LIN {X 0,Y 354.943,Z 301.268,A -85,B 0,C 180,E1 -13486.255,E2 -13486.255} C_VEL
LIN {X 0,Y 354.946,Z 301.27,A -85,B 0,C 180,E1 -13489.735,E2 -13489.735} C_VEL
LIN {X 0,Y 355.073,Z 301.256,A -85,B 0,C 180,E1 -13493.18,E2 -13493.18} C_VEL
LIN {X 0,Y 355.22,Z 301.235,A -85,B 0,C 180,E1 -13497.732,E2 -13497.732} C_VEL
LIN {X 0,Y 355.215,Z 301.234,A -85,B 0,C 180,E1 -13502.268,E2 -13502.268} C_VEL
LIN {X 0,Y 355.075,Z 301.256,A -85,B 0,C 180,E1 -13506.82,E2 -13506.82} C_VEL
LIN {X 0,Y 354.946,Z 301.268,A -85,B 0,C 180,E1 -13510.265,E2 -13510.265} C_VEL
LIN {X 0,Y 354.934,Z 301.269,A -85,B 0,C 180,E1 -13514.019,E2 -13514.019} C_VEL
LIN {X 0,Y 354.881,Z 301.275,A -85,B 0,C 180,E1 -13518.093,E2 -13518.093} C_VEL
LIN {X 0,Y 354.807,Z 301.286,A -85,B 0,C 180,E1 -13522.108,E2 -13522.108} C_VEL
LIN {X 0,Y 354.856,Z 301.278,A -85,B 0,C 180,E1 -13525.831,E2 -13525.831} C_VEL
LIN {X 0,Y 354.8,Z 301.286,A -85,B 0,C 180,E1 -13529.684,E2 -13529.684} C_VEL
LIN {X 0,Y 354.808,Z 301.285,A -85,B 0,C 180,E1 -13533.685,E2 -13533.685} C_VEL
LIN {X 0,Y 354.791,Z 301.292,A -85,B 0,C 180,E1 -13536.46,E2 -13536.46} C_VEL
LIN {X 0,Y 354.818,Z 301.284,A -85,B 0,C 180,E1 -13539.425,E2 -13539.425} C_VEL
LIN {X 0,Y 354.782,Z 301.29,A -85,B 0,C 180,E1 -13542.868,E2 -13542.868} C_VEL
LIN {X 0,Y 354.762,Z 301.294,A -85,B 0,C 180,E1 -13546.105,E2 -13546.105} C_VEL
LIN {X 0,Y 354.783,Z 301.289,A -85,B 0,C 180,E1 -13549.18,E2 -13549.18} C_VEL
LIN {X 0,Y 354.803,Z 301.29,A -85,B 0,C 180,E1 -13552.404,E2 -13552.404} C_VEL
LIN {X 0,Y 354.808,Z 301.286,A -85,B 0,C 180,E1 -13554.942,E2 -13554.942} C_VEL
LIN {X 0,Y 354.791,Z 301.291,A -85,B 0,C 180,E1 -13558.406,E2 -13558.406} C_VEL
LIN {X 0,Y 354.845,Z 301.282,A -85,B 0,C 180,E1 -13561.62,E2 -13561.62} C_VEL
LIN {X 0,Y 354.898,Z 301.28,A -85,B 0,C 180,E1 -13564.174,E2 -13564.174} C_VEL
LIN {X 0,Y 354.845,Z 301.285,A -85,B 0,C 180,E1 -13567.283,E2 -13567.283} C_VEL
LIN {X 0,Y 356.535,Z 305.798,A -85,B 0,C 180,E1 -13567.509,E2 -13567.509} C_VEL
LIN {X 0,Y 362.776,Z 320.32,A -85,B 0,C 180,E1 -13568.226,E2 -13568.226} C_VEL
LIN {X 0,Y 363.979,Z 330.595,A -85,B 0,C 180,E1 -13568.518,E2 -13568.518} C_VEL
LIN {X 0,Y 362.433,Z 414.345,A -85,B 0,C 180,E1 -13570.201,E2 -13570.201} C_VEL
LIN {X 0,Y 361.996,Z 427.668,A -85,B 0,C 180,E1 -13570.693,E2 -13570.693} C_VEL
LIN {X 0,Y 361.185,Z 440.711,A -85,B 0,C 180,E1 -13571.421,E2 -13571.421} C_VEL
LIN {X 0,Y 360.332,Z 451.826,A -85,B 0,C 180,E1 -13572.258,E2 -13572.258} C_VEL
LIN {X 0,Y 359.319,Z 463.137,A -85,B 0,C 180,E1 -13573.356,E2 -13573.356} C_VEL
LIN {X 0,Y 358.318,Z 473.616,A -85,B 0,C 180,E1 -13574.647,E2 -13574.647} C_VEL
LIN {X 0,Y 357.214,Z 482.91,A -85,B 0,C 180,E1 -13576.055,E2 -13576.055} C_VEL
LIN {X 0,Y 356.336,Z 490.521,A -85,B 0,C 180,E1 -13577.471,E2 -13577.471} C_VEL
LIN {X 0,Y 355.47,Z 497.943,A -85,B 0,C 180,E1 -13579.175,E2 -13579.175} C_VEL
LIN {X 0,Y 354.666,Z 503.906,A -85,B 0,C 180,E1 -13580.88,E2 -13580.88} C_VEL
LIN {X 0,Y 354.158,Z 509.234,A -85,B 0,C 180,E1 -13582.848,E2 -13582.848} C_VEL
LIN {X 0,Y 353.853,Z 512.211,A -85,B 0,C 180,E1 -13584.302,E2 -13584.302} C_VEL
LIN {X 0,Y 353.61,Z 514.067,A -85,B 0,C 180,E1 -13585.441,E2 -13585.441} C_VEL
LIN {X 0,Y 353.524,Z 515.48,A -85,B 0,C 180,E1 -13586.582,E2 -13586.582} C_VEL
LIN {X 0,Y 353.413,Z 517.083,A -85,B 0,C 180,E1 -13588.862,E2 -13588.862} C_VEL
LIN {X 0,Y 353.399,Z 517.316,A -85,B 0,C 180,E1 -13590.001,E2 -13590.001} C_VEL
LIN {X 0,Y 353.413,Z 517.125,A -85,B 0,C 180,E1 -13591.141,E2 -13591.141} C_VEL
LIN {X 0,Y 353.52,Z 515.579,A -85,B 0,C 180,E1 -13593.42,E2 -13593.42} C_VEL
LIN {X 0,Y 353.604,Z 514.22,A -85,B 0,C 180,E1 -13594.561,E2 -13594.561} C_VEL
LIN {X 0,Y 353.952,Z 511.354,A -85,B 0,C 180,E1 -13596.271,E2 -13596.271} C_VEL
LIN {X 0,Y 354.266,Z 507.466,A -85,B 0,C 180,E1 -13597.983,E2 -13597.983} C_VEL
LIN {X 0,Y 354.854,Z 502.424,A -85,B 0,C 180,E1 -13599.693,E2 -13599.693} C_VEL
LIN {X 0,Y 355.657,Z 496.064,A -85,B 0,C 180,E1 -13601.398,E2 -13601.398} C_VEL
LIN {X 0,Y 356.581,Z 488.151,A -85,B 0,C 180,E1 -13603.101,E2 -13603.101} C_VEL
LIN {X 0,Y 357.641,Z 480.049,A -85,B 0,C 180,E1 -13604.511,E2 -13604.511} C_VEL
LIN {X 0,Y 358.795,Z 470.095,A -85,B 0,C 180,E1 -13605.917,E2 -13605.917} C_VEL
LIN {X 0,Y 359.629,Z 460.285,A -85,B 0,C 180,E1 -13607.047,E2 -13607.047} C_VEL
LIN {X 0,Y 360.561,Z 449.625,A -85,B 0,C 180,E1 -13608.026,E2 -13608.026} C_VEL
LIN {X 0,Y 361.45,Z 437.916,A -85,B 0,C 180,E1 -13608.861,E2 -13608.861} C_VEL
LIN {X 0,Y 362.145,Z 425.901,A -85,B 0,C 180,E1 -13609.485,E2 -13609.485} C_VEL
LIN {X 0,Y 362.603,Z 412.752,A -85,B 0,C 180,E1 -13609.939,E2 -13609.939} C_VEL
LIN {X 0,Y 363.133,Z 379.152,A -85,B 0,C 180,E1 -13610.626,E2 -13610.626} C_VEL
LIN {X 0,Y 362.558,Z 373.342,A -85,B 0,C 180,E1 -13610.782,E2 -13610.782} C_VEL
LIN {X 0,Y 357.516,Z 354.661,A -85,B 0,C 180,E1 -13611.489,E2 -13611.489} C_VEL
LIN {X 0,Y 357.093,Z 348.851,A -85,B 0,C 180,E1 -13611.64,E2 -13611.64} C_VEL
LIN {X 0,Y 357.337,Z 328.776,A -85,B 0,C 180,E1 -13612.052,E2 -13612.052} C_VEL
LIN {X 0,Y 356.257,Z 322.271,A -85,B 0,C 180,E1 -13612.263,E2 -13612.263} C_VEL
LIN {X 0,Y 347.959,Z 302.988,A -85,B 0,C 180,E1 -13613.254,E2 -13613.254} C_VEL
LIN {X 0,Y 347.823,Z 302.155,A -85,B 0,C 180,E1 -13613.286,E2 -13613.286} C_VEL
LIN {X 0,Y 347.855,Z 302.153,A -85,B 0,C 180,E1 -13617.255,E2 -13617.255} C_VEL
LIN {X 0,Y 347.765,Z 302.164,A -85,B 0,C 180,E1 -13620.347,E2 -13620.347} C_VEL
LIN {X 0,Y 347.749,Z 302.165,A -85,B 0,C 180,E1 -13624.465,E2 -13624.465} C_VEL
LIN {X 0,Y 347.781,Z 302.163,A -85,B 0,C 180,E1 -13627.99,E2 -13627.99} C_VEL
LIN {X 0,Y 347.756,Z 302.167,A -85,B 0,C 180,E1 -13631.831,E2 -13631.831} C_VEL
LIN {X 0,Y 347.772,Z 302.163,A -85,B 0,C 180,E1 -13635.017,E2 -13635.017} C_VEL
LIN {X 0,Y 347.755,Z 302.163,A -85,B 0,C 180,E1 -13638.398,E2 -13638.398} C_VEL
LIN {X 0,Y 347.779,Z 302.161,A -85,B 0,C 180,E1 -13642.012,E2 -13642.012} C_VEL
LIN {X 0,Y 347.75,Z 302.166,A -85,B 0,C 180,E1 -13645.536,E2 -13645.536} C_VEL
LIN {X 0,Y 347.75,Z 302.165,A -85,B 0,C 180,E1 -13648.301,E2 -13648.301} C_VEL
LIN {X 0,Y 347.784,Z 302.165,A -85,B 0,C 180,E1 -13650.988,E2 -13650.988} C_VEL
LIN {X 0,Y 347.836,Z 302.154,A -85,B 0,C 180,E1 -13653.608,E2 -13653.608} C_VEL
LIN {X 0,Y 347.84,Z 302.289,A -85,B 0,C 180,E1 -13657.347,E2 -13657.347} C_VEL
LIN {X 0,Y 348.699,Z 306.937,A -85,B 0,C 180,E1 -13658.715,E2 -13658.715} C_VEL
LIN {X 0,Y 352.108,Z 319.99,A -85,B 0,C 180,E1 -13659.233,E2 -13659.233} C_VEL
LIN {X 0,Y 354.168,Z 331.192,A -85,B 0,C 180,E1 -13659.635,E2 -13659.635} C_VEL
LIN {X 0,Y 351.818,Z 416.062,A -85,B 0,C 180,E1 -13662,E2 -13662} C_VEL
LIN {X 0,Y 351.384,Z 429.687,A -85,B 0,C 180,E1 -13662.616,E2 -13662.616} C_VEL
LIN {X 0,Y 350.662,Z 442.143,A -85,B 0,C 180,E1 -13663.405,E2 -13663.405} C_VEL
LIN {X 0,Y 350.051,Z 454.225,A -85,B 0,C 180,E1 -13664.407,E2 -13664.407} C_VEL
LIN {X 0,Y 349.42,Z 465.515,A -85,B 0,C 180,E1 -13665.587,E2 -13665.587} C_VEL
LIN {X 0,Y 348.563,Z 476.613,A -85,B 0,C 180,E1 -13667.038,E2 -13667.038} C_VEL
LIN {X 0,Y 347.87,Z 486.501,A -85,B 0,C 180,E1 -13668.64,E2 -13668.64} C_VEL
LIN {X 0,Y 347.315,Z 495.155,A -85,B 0,C 180,E1 -13670.39,E2 -13670.39} C_VEL
LIN {X 0,Y 346.876,Z 502.131,A -85,B 0,C 180,E1 -13672.139,E2 -13672.139} C_VEL
LIN {X 0,Y 346.533,Z 507.828,A -85,B 0,C 180,E1 -13673.954,E2 -13673.954} C_VEL
LIN {X 0,Y 346.411,Z 512.511,A -85,B 0,C 180,E1 -13675.928,E2 -13675.928} C_VEL
LIN {X 0,Y 346.281,Z 515.485,A -85,B 0,C 180,E1 -13677.674,E2 -13677.674} C_VEL
LIN {X 0,Y 346.265,Z 516.905,A -85,B 0,C 180,E1 -13678.837,E2 -13678.837} C_VEL
LIN {X 0,Y 346.291,Z 517.875,A -85,B 0,C 180,E1 -13680,E2 -13680} C_VEL
LIN {X 0,Y 346.374,Z 518.383,A -85,B 0,C 180,E1 -13681.163,E2 -13681.163} C_VEL
LIN {X 0,Y 346.512,Z 518.476,A -85,B 0,C 180,E1 -13682.325,E2 -13682.325} C_VEL
LIN {X 0,Y 346.709,Z 518.149,A -85,B 0,C 180,E1 -13683.486,E2 -13683.486} C_VEL
LIN {X 0,Y 346.782,Z 517.364,A -85,B 0,C 180,E1 -13684.65,E2 -13684.65} C_VEL
LIN {X 0,Y 346.874,Z 516.16,A -85,B 0,C 180,E1 -13685.814,E2 -13685.814} C_VEL
LIN {X 0,Y 347.646,Z 512.916,A -85,B 0,C 180,E1 -13687.864,E2 -13687.864} C_VEL
LIN {X 0,Y 348.502,Z 508.27,A -85,B 0,C 180,E1 -13689.87,E2 -13689.87} C_VEL
LIN {X 0,Y 349.62,Z 501.96,A -85,B 0,C 180,E1 -13691.891,E2 -13691.891} C_VEL
LIN {X 0,Y 350.753,Z 495.084,A -85,B 0,C 180,E1 -13693.617,E2 -13693.617} C_VEL
LIN {X 0,Y 352.112,Z 486.474,A -85,B 0,C 180,E1 -13695.335,E2 -13695.335} C_VEL
LIN {X 0,Y 353.615,Z 477.681,A -85,B 0,C 180,E1 -13696.749,E2 -13696.749} C_VEL
LIN {X 0,Y 355.127,Z 467.571,A -85,B 0,C 180,E1 -13698.083,E2 -13698.083} C_VEL
LIN {X 0,Y 356.807,Z 454.872,A -85,B 0,C 180,E1 -13699.413,E2 -13699.413} C_VEL
LIN {X 0,Y 358.181,Z 442.944,A -85,B 0,C 180,E1 -13700.382,E2 -13700.382} C_VEL
LIN {X 0,Y 359.347,Z 429.73,A -85,B 0,C 180,E1 -13701.212,E2 -13701.212} C_VEL
LIN {X 0,Y 360.302,Z 416.514,A -85,B 0,C 180,E1 -13701.791,E2 -13701.791} C_VEL
LIN {X 0,Y 365.349,Z 340.859,A -85,B 0,C 180,E1 -13704.251,E2 -13704.251} C_VEL
LIN {X 0,Y 363.993,Z 337.298,A -85,B 0,C 180,E1 -13704.591,E2 -13704.591} C_VEL
LIN {X 0,Y 358.725,Z 326.902,A -85,B 0,C 180,E1 -13705.835,E2 -13705.835} C_VEL
LIN {X 0,Y 353.588,Z 318.534,A -85,B 0,C 180,E1 -13707.102,E2 -13707.102} C_VEL
LIN {X 0,Y 351.324,Z 314.748,A -85,B 0,C 180,E1 -13707.724,E2 -13707.724} C_VEL
LIN {X 0,Y 350.188,Z 310.445,A -85,B 0,C 180,E1 -13710.346,E2 -13710.346} C_VEL
LIN {X 0,Y 349.155,Z 306.963,A -85,B 0,C 180,E1 -13712.92,E2 -13712.92} C_VEL
LIN {X 0,Y 348.281,Z 304.055,A -85,B 0,C 180,E1 -13715.817,E2 -13715.817} C_VEL
LIN {X 0,Y 347.734,Z 302.169,A -85,B 0,C 180,E1 -13718.795,E2 -13718.795} C_VEL
LIN {X 0,Y 347.743,Z 302.169,A -85,B 0,C 180,E1 -13721.831,E2 -13721.831} C_VEL
LIN {X 0,Y 347.742,Z 302.182,A -85,B 0,C 180,E1 -13725.42,E2 -13725.42} C_VEL
LIN {X 0,Y 348.287,Z 304.196,A -85,B 0,C 180,E1 -13728.298,E2 -13728.298} C_VEL
LIN {X 0,Y 348.856,Z 305.831,A -85,B 0,C 180,E1 -13729.955,E2 -13729.955} C_VEL
LIN {X 0,Y 350.413,Z 310.427,A -85,B 0,C 180,E1 -13733.346,E2 -13733.346} C_VEL
LIN {X 0,Y 351.765,Z 315.246,A -85,B 0,C 180,E1 -13735.983,E2 -13735.983} C_VEL
LIN {X 0,Y 353.418,Z 321.647,A -85,B 0,C 180,E1 -13738.866,E2 -13738.866} C_VEL
LIN {X 0,Y 354.923,Z 328.994,A -85,B 0,C 180,E1 -13741.624,E2 -13741.624} C_VEL
LIN {X 0,Y 355.421,Z 333.185,A -85,B 0,C 180,E1 -13743.008,E2 -13743.008} C_VEL
LIN {X 0,Y 358.864,Z 346.581,A -85,B 0,C 180,E1 -13744.17,E2 -13744.17} C_VEL
LIN {X 0,Y 361.513,Z 360.04,A -85,B 0,C 180,E1 -13745.139,E2 -13745.139} C_VEL
LIN {X 0,Y 363.058,Z 371.025,A -85,B 0,C 180,E1 -13745.804,E2 -13745.804} C_VEL
LIN {X 0,Y 363.51,Z 377.914,A -85,B 0,C 180,E1 -13746.146,E2 -13746.146} C_VEL
LIN {X 0,Y 359.161,Z 446.637,A -85,B 0,C 180,E1 -13748.362,E2 -13748.362} C_VEL
LIN {X 0,Y 357.866,Z 460.11,A -85,B 0,C 180,E1 -13748.997,E2 -13748.997} C_VEL
LIN {X 0,Y 356.387,Z 472.712,A -85,B 0,C 180,E1 -13749.811,E2 -13749.811} C_VEL
LIN {X 0,Y 354.63,Z 485.801,A -85,B 0,C 180,E1 -13750.913,E2 -13750.913} C_VEL
LIN {X 0,Y 352.739,Z 498.651,A -85,B 0,C 180,E1 -13752.31,E2 -13752.31} C_VEL
LIN {X 0,Y 351.199,Z 508.989,A -85,B 0,C 180,E1 -13753.729,E2 -13753.729} C_VEL
LIN {X 0,Y 349.796,Z 517.581,A -85,B 0,C 180,E1 -13755.156,E2 -13755.156} C_VEL
LIN {X 0,Y 348.612,Z 526.071,A -85,B 0,C 180,E1 -13756.89,E2 -13756.89} C_VEL
LIN {X 0,Y 347.626,Z 532.987,A -85,B 0,C 180,E1 -13758.63,E2 -13758.63} C_VEL
LIN {X 0,Y 346.843,Z 539.297,A -85,B 0,C 180,E1 -13760.67,E2 -13760.67} C_VEL
LIN {X 0,Y 346.405,Z 543.453,A -85,B 0,C 180,E1 -13762.421,E2 -13762.421} C_VEL
LIN {X 0,Y 346.23,Z 546.523,A -85,B 0,C 180,E1 -13764.174,E2 -13764.174} C_VEL
LIN {X 0,Y 346.181,Z 548.006,A -85,B 0,C 180,E1 -13765.341,E2 -13765.341} C_VEL
LIN {X 0,Y 346.167,Z 549.058,A -85,B 0,C 180,E1 -13766.507,E2 -13766.507} C_VEL
LIN {X 0,Y 346.159,Z 549.629,A -85,B 0,C 180,E1 -13767.672,E2 -13767.672} C_VEL
LIN {X 0,Y 346.29,Z 549.774,A -85,B 0,C 180,E1 -13768.836,E2 -13768.836} C_VEL
LIN {X 0,Y 346.36,Z 549.487,A -85,B 0,C 180,E1 -13769.999,E2 -13769.999} C_VEL
LIN {X 0,Y 346.289,Z 547.742,A -85,B 0,C 180,E1 -13772.325,E2 -13772.325} C_VEL
LIN {X 0,Y 346.22,Z 546.705,A -85,B 0,C 180,E1 -13773.49,E2 -13773.49} C_VEL
LIN {X 0,Y 346.251,Z 545.261,A -85,B 0,C 180,E1 -13774.656,E2 -13774.656} C_VEL
LIN {X 0,Y 346.281,Z 542.259,A -85,B 0,C 180,E1 -13776.407,E2 -13776.407} C_VEL
LIN {X 0,Y 346.488,Z 538.188,A -85,B 0,C 180,E1 -13778.161,E2 -13778.161} C_VEL
LIN {X 0,Y 346.933,Z 531.911,A -85,B 0,C 180,E1 -13780.209,E2 -13780.209} C_VEL
LIN {X 0,Y 347.597,Z 525.071,A -85,B 0,C 180,E1 -13781.96,E2 -13781.96} C_VEL
LIN {X 0,Y 348.436,Z 518.09,A -85,B 0,C 180,E1 -13783.411,E2 -13783.411} C_VEL
LIN {X 0,Y 349.454,Z 509.07,A -85,B 0,C 180,E1 -13784.947,E2 -13784.947} C_VEL
LIN {X 0,Y 350.467,Z 499.204,A -85,B 0,C 180,E1 -13786.303,E2 -13786.303} C_VEL
LIN {X 0,Y 351.59,Z 488.855,A -85,B 0,C 180,E1 -13787.447,E2 -13787.447} C_VEL
LIN {X 0,Y 352.712,Z 477.474,A -85,B 0,C 180,E1 -13788.439,E2 -13788.439} C_VEL
LIN {X 0,Y 353.77,Z 464.4,A -85,B 0,C 180,E1 -13789.284,E2 -13789.284} C_VEL
LIN {X 0,Y 354.594,Z 452.101,A -85,B 0,C 180,E1 -13789.84,E2 -13789.84} C_VEL
LIN {X 0,Y 355.014,Z 439.719,A -85,B 0,C 180,E1 -13790.193,E2 -13790.193} C_VEL
LIN {X 0,Y 356.114,Z 374.524,A -85,B 0,C 180,E1 -13791.499,E2 -13791.499} C_VEL
LIN {X 0,Y 350.634,Z 335.789,A -85,B 0,C 180,E1 -13792.683,E2 -13792.683} C_VEL
LIN {X 0,Y 350.215,Z 333.047,A -85,B 0,C 180,E1 -13792.779,E2 -13792.779} C_VEL
LIN {X 0,Y 351.339,Z 321.609,A -85,B 0,C 180,E1 -13795.405,E2 -13795.405} C_VEL
LIN {X 0,Y 350.883,Z 317.2,A -85,B 0,C 180,E1 -13796.464,E2 -13796.464} C_VEL
LIN {X 0,Y 348.529,Z 305.733,A -85,B 0,C 180,E1 -13799.339,E2 -13799.339} C_VEL
LIN {X 0,Y 347.809,Z 302.162,A -85,B 0,C 180,E1 -13800.254,E2 -13800.254} C_VEL
LIN {X 0,Y 347.741,Z 302.168,A -85,B 0,C 180,E1 -13804.463,E2 -13804.463} C_VEL
LIN {X 0,Y 347.767,Z 302.168,A -85,B 0,C 180,E1 -13807.987,E2 -13807.987} C_VEL
LIN {X 0,Y 347.743,Z 302.17,A -85,B 0,C 180,E1 -13811.83,E2 -13811.83} C_VEL
LIN {X 0,Y 347.7,Z 302.17,A -85,B 0,C 180,E1 -13815.026,E2 -13815.026} C_VEL
LIN {X 0,Y 347.735,Z 302.167,A -85,B 0,C 180,E1 -13818.398,E2 -13818.398} C_VEL
LIN {X 0,Y 347.75,Z 302.164,A -85,B 0,C 180,E1 -13822.678,E2 -13822.678} C_VEL
LIN {X 0,Y 347.741,Z 302.169,A -85,B 0,C 180,E1 -13825.955,E2 -13825.955} C_VEL
LIN {X 0,Y 347.73,Z 302.172,A -85,B 0,C 180,E1 -13829.65,E2 -13829.65} C_VEL
LIN {X 0,Y 347.729,Z 302.172,A -85,B 0,C 180,E1 -13833.599,E2 -13833.599} C_VEL
LIN {X 0,Y 347.744,Z 302.166,A -85,B 0,C 180,E1 -13836.159,E2 -13836.159} C_VEL
LIN {X 0,Y 347.791,Z 302.16,A -85,B 0,C 180,E1 -13839.908,E2 -13839.908} C_VEL
LIN {X 0,Y 347.823,Z 302.158,A -85,B 0,C 180,E1 -13843.568,E2 -13843.568} C_VEL
LIN {X 0,Y 347.88,Z 302.152,A -85,B 0,C 180,E1 -13847.16,E2 -13847.16} C_VEL
LIN {X 0,Y 347.926,Z 302.143,A -85,B 0,C 180,E1 -13850.7,E2 -13850.7} C_VEL
LIN {X 0,Y 348.025,Z 302.125,A -85,B 0,C 180,E1 -13854.205,E2 -13854.205} C_VEL
LIN {X 0,Y 348.181,Z 302.111,A -85,B 0,C 180,E1 -13857.686,E2 -13857.686} C_VEL
LIN {X 0,Y 348.13,Z 302.122,A -85,B 0,C 180,E1 -13861.157,E2 -13861.157} C_VEL
LIN {X 0,Y 348.176,Z 302.111,A -85,B 0,C 180,E1 -13862.314,E2 -13862.314} C_VEL
LIN {X 0,Y 348.043,Z 302.133,A -85,B 0,C 180,E1 -13866.959,E2 -13866.959} C_VEL
LIN {X 0,Y 347.887,Z 302.148,A -85,B 0,C 180,E1 -13870.476,E2 -13870.476} C_VEL
LIN {X 0,Y 347.89,Z 302.147,A -85,B 0,C 180,E1 -13874.15,E2 -13874.15} C_VEL
LIN {X 0,Y 347.821,Z 302.155,A -85,B 0,C 180,E1 -13878.26,E2 -13878.26} C_VEL
LIN {X 0,Y 347.759,Z 302.163,A -85,B 0,C 180,E1 -13881.627,E2 -13881.627} C_VEL
LIN {X 0,Y 347.785,Z 302.161,A -85,B 0,C 180,E1 -13885.111,E2 -13885.111} C_VEL
LIN {X 0,Y 347.75,Z 302.167,A -85,B 0,C 180,E1 -13889.015,E2 -13889.015} C_VEL
LIN {X 0,Y 347.726,Z 302.169,A -85,B 0,C 180,E1 -13893.073,E2 -13893.073} C_VEL
LIN {X 0,Y 347.764,Z 302.164,A -85,B 0,C 180,E1 -13896.066,E2 -13896.066} C_VEL
LIN {X 0,Y 347.746,Z 302.168,A -85,B 0,C 180,E1 -13898.794,E2 -13898.794} C_VEL
LIN {X 0,Y 347.744,Z 302.166,A -85,B 0,C 180,E1 -13901.831,E2 -13901.831} C_VEL
LIN {X 0,Y 347.7,Z 302.172,A -85,B 0,C 180,E1 -13905.028,E2 -13905.028} C_VEL
LIN {X 0,Y 347.746,Z 302.171,A -85,B 0,C 180,E1 -13908.398,E2 -13908.398} C_VEL
LIN {X 0,Y 347.769,Z 302.164,A -85,B 0,C 180,E1 -13912.013,E2 -13912.013} C_VEL
LIN {X 0,Y 347.741,Z 302.166,A -85,B 0,C 180,E1 -13915.537,E2 -13915.537} C_VEL
LIN {X 0,Y 347.742,Z 302.169,A -85,B 0,C 180,E1 -13918.302,E2 -13918.302} C_VEL
LIN {X 0,Y 347.776,Z 302.161,A -85,B 0,C 180,E1 -13920.989,E2 -13920.989} C_VEL
LIN {X 0,Y 347.829,Z 302.156,A -85,B 0,C 180,E1 -13923.609,E2 -13923.609} C_VEL
LIN {X 0,Y 347.809,Z 302.162,A -85,B 0,C 180,E1 -13926.818,E2 -13926.818} C_VEL
LIN {X 0,Y 349.299,Z 306.157,A -85,B 0,C 180,E1 -13927.019,E2 -13927.019} C_VEL
LIN {X 0,Y 356.462,Z 322.892,A -85,B 0,C 180,E1 -13927.871,E2 -13927.871} C_VEL
LIN {X 0,Y 357.407,Z 331.113,A -85,B 0,C 180,E1 -13928.109,E2 -13928.109} C_VEL
LIN {X 0,Y 355.77,Z 414.603,A -85,B 0,C 180,E1 -13929.814,E2 -13929.814} C_VEL
LIN {X 0,Y 355.322,Z 427.956,A -85,B 0,C 180,E1 -13930.315,E2 -13930.315} C_VEL
LIN {X 0,Y 354.49,Z 441.01,A -85,B 0,C 180,E1 -13931.057,E2 -13931.057} C_VEL
LIN {X 0,Y 353.602,Z 452.131,A -85,B 0,C 180,E1 -13931.909,E2 -13931.909} C_VEL
LIN {X 0,Y 352.649,Z 462.317,A -85,B 0,C 180,E1 -13932.9,E2 -13932.9} C_VEL
LIN {X 0,Y 351.631,Z 472.892,A -85,B 0,C 180,E1 -13934.199,E2 -13934.199} C_VEL
LIN {X 0,Y 350.343,Z 483.223,A -85,B 0,C 180,E1 -13935.776,E2 -13935.776} C_VEL
LIN {X 0,Y 349.419,Z 490.836,A -85,B 0,C 180,E1 -13937.219,E2 -13937.219} C_VEL
LIN {X 0,Y 348.5,Z 498.259,A -85,B 0,C 180,E1 -13938.956,E2 -13938.956} C_VEL
LIN {X 0,Y 347.678,Z 504.222,A -85,B 0,C 180,E1 -13940.695,E2 -13940.695} C_VEL
LIN {X 0,Y 347.178,Z 508.93,A -85,B 0,C 180,E1 -13942.441,E2 -13942.441} C_VEL
LIN {X 0,Y 346.789,Z 512.528,A -85,B 0,C 180,E1 -13944.185,E2 -13944.185} C_VEL
LIN {X 0,Y 346.55,Z 514.383,A -85,B 0,C 180,E1 -13945.348,E2 -13945.348} C_VEL
LIN {X 0,Y 346.437,Z 515.798,A -85,B 0,C 180,E1 -13946.512,E2 -13946.512} C_VEL
LIN {X 0,Y 346.321,Z 517.4,A -85,B 0,C 180,E1 -13948.838,E2 -13948.838} C_VEL
LIN {X 0,Y 346.321,Z 517.633,A -85,B 0,C 180,E1 -13950.001,E2 -13950.001} C_VEL
LIN {X 0,Y 346.321,Z 517.441,A -85,B 0,C 180,E1 -13951.164,E2 -13951.164} C_VEL
LIN {X 0,Y 346.434,Z 515.895,A -85,B 0,C 180,E1 -13953.49,E2 -13953.49} C_VEL
LIN {X 0,Y 346.546,Z 514.535,A -85,B 0,C 180,E1 -13954.654,E2 -13954.654} C_VEL
LIN {X 0,Y 346.939,Z 511.247,A -85,B 0,C 180,E1 -13956.605,E2 -13956.605} C_VEL
LIN {X 0,Y 347.424,Z 506.215,A -85,B 0,C 180,E1 -13958.728,E2 -13958.728} C_VEL
LIN {X 0,Y 348.165,Z 500.773,A -85,B 0,C 180,E1 -13960.468,E2 -13960.468} C_VEL
LIN {X 0,Y 348.999,Z 493.95,A -85,B 0,C 180,E1 -13962.208,E2 -13962.208} C_VEL
LIN {X 0,Y 350.082,Z 485.393,A -85,B 0,C 180,E1 -13963.941,E2 -13963.941} C_VEL
LIN {X 0,Y 351.24,Z 476.623,A -85,B 0,C 180,E1 -13965.375,E2 -13965.375} C_VEL
LIN {X 0,Y 352.234,Z 466.935,A -85,B 0,C 180,E1 -13966.675,E2 -13966.675} C_VEL
LIN {X 0,Y 353.256,Z 456.315,A -85,B 0,C 180,E1 -13967.812,E2 -13967.812} C_VEL
LIN {X 0,Y 354.283,Z 444.448,A -85,B 0,C 180,E1 -13968.807,E2 -13968.807} C_VEL
LIN {X 0,Y 355.107,Z 432.028,A -85,B 0,C 180,E1 -13969.587,E2 -13969.587} C_VEL
LIN {X 0,Y 355.725,Z 418.881,A -85,B 0,C 180,E1 -13970.153,E2 -13970.153} C_VEL
LIN {X 0,Y 356.047,Z 404.979,A -85,B 0,C 180,E1 -13970.511,E2 -13970.511} C_VEL
LIN {X 0,Y 357.093,Z 348.851,A -85,B 0,C 180,E1 -13971.64,E2 -13971.64} C_VEL
LIN {X 0,Y 356.741,Z 342.979,A -85,B 0,C 180,E1 -13971.788,E2 -13971.788} C_VEL
LIN {X 0,Y 355.451,Z 337.283,A -85,B 0,C 180,E1 -13971.994,E2 -13971.994} C_VEL
LIN {X 0,Y 354.215,Z 333.617,A -85,B 0,C 180,E1 -13972.154,E2 -13972.154} C_VEL
LIN {X 0,Y 347.775,Z 319.399,A -85,B 0,C 180,E1 -13972.904,E2 -13972.904} C_VEL
LIN {X 0,Y 340.811,Z 303.416,A -85,B 0,C 180,E1 -13973.766,E2 -13973.766} C_VEL
LIN {X 0,Y 340.752,Z 303.04,A -85,B 0,C 180,E1 -13973.827,E2 -13973.827} C_VEL
LIN {X 0,Y 340.781,Z 303.036,A -85,B 0,C 180,E1 -13977.526,E2 -13977.526} C_VEL
LIN {X 0,Y 340.773,Z 303.038,A -85,B 0,C 180,E1 -13979.98,E2 -13979.98} C_VEL
LIN {X 0,Y 340.699,Z 303.047,A -85,B 0,C 180,E1 -13983.847,E2 -13983.847} C_VEL
LIN {X 0,Y 340.711,Z 303.041,A -85,B 0,C 180,E1 -13986.742,E2 -13986.742} C_VEL
LIN {X 0,Y 340.693,Z 303.045,A -85,B 0,C 180,E1 -13990.248,E2 -13990.248} C_VEL
LIN {X 0,Y 340.67,Z 303.047,A -85,B 0,C 180,E1 -13993.776,E2 -13993.776} C_VEL
LIN {X 0,Y 340.683,Z 303.043,A -85,B 0,C 180,E1 -13997.096,E2 -13997.096} C_VEL
LIN {X 0,Y 340.704,Z 303.043,A -85,B 0,C 180,E1 -14000.248,E2 -14000.248} C_VEL
LIN {X 0,Y 340.715,Z 303.042,A -85,B 0,C 180,E1 -14003.56,E2 -14003.56} C_VEL
LIN {X 0,Y 340.698,Z 303.043,A -85,B 0,C 180,E1 -14006.154,E2 -14006.154} C_VEL
LIN {X 0,Y 340.747,Z 303.036,A -85,B 0,C 180,E1 -14010.33,E2 -14010.33} C_VEL
LIN {X 0,Y 340.808,Z 303.033,A -85,B 0,C 180,E1 -14013.02,E2 -14013.02} C_VEL
LIN {X 0,Y 340.763,Z 303.04,A -85,B 0,C 180,E1 -14017.071,E2 -14017.071} C_VEL
LIN {X 0,Y 340.793,Z 303.186,A -85,B 0,C 180,E1 -14017.215,E2 -14017.215} C_VEL
LIN {X 0,Y 341.55,Z 307.197,A -85,B 0,C 180,E1 -14018.416,E2 -14018.416} C_VEL
LIN {X 0,Y 345.363,Z 321.819,A -85,B 0,C 180,E1 -14019.02,E2 -14019.02} C_VEL
LIN {X 0,Y 347.228,Z 332.491,A -85,B 0,C 180,E1 -14019.41,E2 -14019.41} C_VEL
LIN {X 0,Y 344.826,Z 416.133,A -85,B 0,C 180,E1 -14021.815,E2 -14021.815} C_VEL
LIN {X 0,Y 344.323,Z 430.424,A -85,B 0,C 180,E1 -14022.478,E2 -14022.478} C_VEL
LIN {X 0,Y 343.58,Z 443.706,A -85,B 0,C 180,E1 -14023.359,E2 -14023.359} C_VEL
LIN {X 0,Y 342.935,Z 455.86,A -85,B 0,C 180,E1 -14024.412,E2 -14024.412} C_VEL
LIN {X 0,Y 342.279,Z 466.584,A -85,B 0,C 180,E1 -14025.584,E2 -14025.584} C_VEL
LIN {X 0,Y 341.435,Z 477.584,A -85,B 0,C 180,E1 -14027.065,E2 -14027.065} C_VEL
LIN {X 0,Y 340.751,Z 487.344,A -85,B 0,C 180,E1 -14028.7,E2 -14028.7} C_VEL
LIN {X 0,Y 340.175,Z 495.926,A -85,B 0,C 180,E1 -14030.486,E2 -14030.486} C_VEL
LIN {X 0,Y 339.734,Z 502.818,A -85,B 0,C 180,E1 -14032.272,E2 -14032.272} C_VEL
LIN {X 0,Y 339.442,Z 508.263,A -85,B 0,C 180,E1 -14034.058,E2 -14034.058} C_VEL
LIN {X 0,Y 339.342,Z 512.479,A -85,B 0,C 180,E1 -14035.843,E2 -14035.843} C_VEL
LIN {X 0,Y 339.188,Z 515.581,A -85,B 0,C 180,E1 -14037.625,E2 -14037.625} C_VEL
LIN {X 0,Y 339.167,Z 517.065,A -85,B 0,C 180,E1 -14038.813,E2 -14038.813} C_VEL
LIN {X 0,Y 339.196,Z 518.127,A -85,B 0,C 180,E1 -14040,E2 -14040} C_VEL
LIN {X 0,Y 339.284,Z 518.72,A -85,B 0,C 180,E1 -14041.187,E2 -14041.187} C_VEL
LIN {X 0,Y 339.428,Z 518.874,A -85,B 0,C 180,E1 -14042.373,E2 -14042.373} C_VEL
LIN {X 0,Y 339.629,Z 518.614,A -85,B 0,C 180,E1 -14043.559,E2 -14043.559} C_VEL
LIN {X 0,Y 339.716,Z 517.938,A -85,B 0,C 180,E1 -14044.747,E2 -14044.747} C_VEL
LIN {X 0,Y 339.847,Z 516.798,A -85,B 0,C 180,E1 -14045.935,E2 -14045.935} C_VEL
LIN {X 0,Y 340.617,Z 513.833,A -85,B 0,C 180,E1 -14047.943,E2 -14047.943} C_VEL
LIN {X 0,Y 341.577,Z 509.232,A -85,B 0,C 180,E1 -14050.072,E2 -14050.072} C_VEL
LIN {X 0,Y 342.763,Z 503.078,A -85,B 0,C 180,E1 -14052.132,E2 -14052.132} C_VEL
LIN {X 0,Y 343.984,Z 496.39,A -85,B 0,C 180,E1 -14053.89,E2 -14053.89} C_VEL
LIN {X 0,Y 345.43,Z 488.056,A -85,B 0,C 180,E1 -14055.639,E2 -14055.639} C_VEL
LIN {X 0,Y 347.003,Z 479.519,A -85,B 0,C 180,E1 -14057.078,E2 -14057.078} C_VEL
LIN {X 0,Y 348.818,Z 468.463,A -85,B 0,C 180,E1 -14058.594,E2 -14058.594} C_VEL
LIN {X 0,Y 350.577,Z 456.134,A -85,B 0,C 180,E1 -14059.926,E2 -14059.926} C_VEL
LIN {X 0,Y 352.066,Z 444.56,A -85,B 0,C 180,E1 -14060.905,E2 -14060.905} C_VEL
LIN {X 0,Y 353.396,Z 430.593,A -85,B 0,C 180,E1 -14061.817,E2 -14061.817} C_VEL
LIN {X 0,Y 354.486,Z 416.865,A -85,B 0,C 180,E1 -14062.436,E2 -14062.436} C_VEL
LIN {X 0,Y 359.794,Z 342.877,A -85,B 0,C 180,E1 -14064.928,E2 -14064.928} C_VEL
LIN {X 0,Y 355.255,Z 333.467,A -85,B 0,C 180,E1 -14066.062,E2 -14066.062} C_VEL
LIN {X 0,Y 350.028,Z 324.309,A -85,B 0,C 180,E1 -14067.434,E2 -14067.434} C_VEL
LIN {X 0,Y 346.681,Z 319.373,A -85,B 0,C 180,E1 -14068.349,E2 -14068.349} C_VEL
LIN {X 0,Y 344.414,Z 315.634,A -85,B 0,C 180,E1 -14069.061,E2 -14069.061} C_VEL
LIN {X 0,Y 343.228,Z 311.23,A -85,B 0,C 180,E1 -14072.167,E2 -14072.167} C_VEL
LIN {X 0,Y 342.253,Z 308.155,A -85,B 0,C 180,E1 -14075.097,E2 -14075.097} C_VEL
LIN {X 0,Y 341.631,Z 305.781,A -85,B 0,C 180,E1 -14078.579,E2 -14078.579} C_VEL
LIN {X 0,Y 341.266,Z 305.082,A -85,B 0,C 180,E1 -14082.149,E2 -14082.149} C_VEL
LIN {X 0,Y 341.661,Z 305.917,A -85,B 0,C 180,E1 -14085.621,E2 -14085.621} C_VEL
LIN {X 0,Y 342.325,Z 308.368,A -85,B 0,C 180,E1 -14088.93,E2 -14088.93} C_VEL
LIN {X 0,Y 343.588,Z 312.122,A -85,B 0,C 180,E1 -14092.146,E2 -14092.146} C_VEL
LIN {X 0,Y 344.779,Z 316.06,A -85,B 0,C 180,E1 -14094.624,E2 -14094.624} C_VEL
LIN {X 0,Y 346.256,Z 321.648,A -85,B 0,C 180,E1 -14097.46,E2 -14097.46} C_VEL
LIN {X 0,Y 347.404,Z 326.687,A -85,B 0,C 180,E1 -14099.618,E2 -14099.618} C_VEL
LIN {X 0,Y 348.545,Z 332.551,A -85,B 0,C 180,E1 -14101.792,E2 -14101.792} C_VEL
LIN {X 0,Y 350.974,Z 338.223,A -85,B 0,C 180,E1 -14102.521,E2 -14102.521} C_VEL
LIN {X 0,Y 354.022,Z 350.788,A -85,B 0,C 180,E1 -14103.641,E2 -14103.641} C_VEL
LIN {X 0,Y 356.472,Z 364.409,A -85,B 0,C 180,E1 -14104.642,E2 -14104.642} C_VEL
LIN {X 0,Y 357.846,Z 376.762,A -85,B 0,C 180,E1 -14105.378,E2 -14105.378} C_VEL
LIN {X 0,Y 357.302,Z 386.711,A -85,B 0,C 180,E1 -14105.739,E2 -14105.739} C_VEL
LIN {X 0,Y 353.188,Z 446.882,A -85,B 0,C 180,E1 -14107.746,E2 -14107.746} C_VEL
LIN {X 0,Y 351.659,Z 461.131,A -85,B 0,C 180,E1 -14108.454,E2 -14108.454} C_VEL
LIN {X 0,Y 350.134,Z 473.345,A -85,B 0,C 180,E1 -14109.281,E2 -14109.281} C_VEL
LIN {X 0,Y 348.497,Z 484.694,A -85,B 0,C 180,E1 -14110.257,E2 -14110.257} C_VEL
LIN {X 0,Y 346.676,Z 496.429,A -85,B 0,C 180,E1 -14111.532,E2 -14111.532} C_VEL
LIN {X 0,Y 345.107,Z 506.098,A -85,B 0,C 180,E1 -14112.824,E2 -14112.824} C_VEL
LIN {X 0,Y 343.427,Z 515.259,A -85,B 0,C 180,E1 -14114.292,E2 -14114.292} C_VEL
LIN {X 0,Y 342.167,Z 523.94,A -85,B 0,C 180,E1 -14116.033,E2 -14116.033} C_VEL
LIN {X 0,Y 340.941,Z 531.149,A -85,B 0,C 180,E1 -14117.801,E2 -14117.801} C_VEL
LIN {X 0,Y 340.001,Z 537.836,A -85,B 0,C 180,E1 -14119.88,E2 -14119.88} C_VEL
LIN {X 0,Y 339.513,Z 542.243,A -85,B 0,C 180,E1 -14121.667,E2 -14121.667} C_VEL
LIN {X 0,Y 339.255,Z 544.54,A -85,B 0,C 180,E1 -14122.859,E2 -14122.859} C_VEL
LIN {X 0,Y 339.136,Z 546.478,A -85,B 0,C 180,E1 -14124.109,E2 -14124.109} C_VEL
LIN {X 0,Y 339.084,Z 547.826,A -85,B 0,C 180,E1 -14125.243,E2 -14125.243} C_VEL
LIN {X 0,Y 339.09,Z 548.779,A -85,B 0,C 180,E1 -14126.434,E2 -14126.434} C_VEL
LIN {X 0,Y 339.069,Z 549.289,A -85,B 0,C 180,E1 -14127.623,E2 -14127.623} C_VEL
LIN {X 0,Y 339.195,Z 549.382,A -85,B 0,C 180,E1 -14128.812,E2 -14128.812} C_VEL
LIN {X 0,Y 339.299,Z 549.033,A -85,B 0,C 180,E1 -14129.999,E2 -14129.999} C_VEL
LIN {X 0,Y 339.189,Z 547.41,A -85,B 0,C 180,E1 -14132.374,E2 -14132.374} C_VEL
LIN {X 0,Y 339.141,Z 546.388,A -85,B 0,C 180,E1 -14133.563,E2 -14133.563} C_VEL
LIN {X 0,Y 339.146,Z 544.942,A -85,B 0,C 180,E1 -14134.754,E2 -14134.754} C_VEL
LIN {X 0,Y 339.202,Z 541.94,A -85,B 0,C 180,E1 -14136.542,E2 -14136.542} C_VEL
LIN {X 0,Y 339.419,Z 537.87,A -85,B 0,C 180,E1 -14138.333,E2 -14138.333} C_VEL
LIN {X 0,Y 339.902,Z 531.592,A -85,B 0,C 180,E1 -14140.422,E2 -14140.422} C_VEL
LIN {X 0,Y 340.63,Z 524.754,A -85,B 0,C 180,E1 -14142.208,E2 -14142.208} C_VEL
LIN {X 0,Y 341.478,Z 517.773,A -85,B 0,C 180,E1 -14143.69,E2 -14143.69} C_VEL
LIN {X 0,Y 342.539,Z 508.754,A -85,B 0,C 180,E1 -14145.256,E2 -14145.256} C_VEL
LIN {X 0,Y 343.611,Z 498.891,A -85,B 0,C 180,E1 -14146.638,E2 -14146.638} C_VEL
LIN {X 0,Y 344.812,Z 488.547,A -85,B 0,C 180,E1 -14147.801,E2 -14147.801} C_VEL
LIN {X 0,Y 345.985,Z 477.172,A -85,B 0,C 180,E1 -14148.811,E2 -14148.811} C_VEL
LIN {X 0,Y 346.987,Z 465.387,A -85,B 0,C 180,E1 -14149.599,E2 -14149.599} C_VEL
LIN {X 0,Y 347.879,Z 452.716,A -85,B 0,C 180,E1 -14150.201,E2 -14150.201} C_VEL
LIN {X 0,Y 348.349,Z 439.489,A -85,B 0,C 180,E1 -14150.596,E2 -14150.596} C_VEL
LIN {X 0,Y 349.508,Z 375.231,A -85,B 0,C 180,E1 -14151.906,E2 -14151.906} C_VEL
LIN {X 0,Y 344.087,Z 336.981,A -85,B 0,C 180,E1 -14153.108,E2 -14153.108} C_VEL
LIN {X 0,Y 343.274,Z 331.935,A -85,B 0,C 180,E1 -14153.285,E2 -14153.285} C_VEL
LIN {X 0,Y 344.305,Z 321.595,A -85,B 0,C 180,E1 -14155.715,E2 -14155.715} C_VEL
LIN {X 0,Y 343.122,Z 314.712,A -85,B 0,C 180,E1 -14157.441,E2 -14157.441} C_VEL
LIN {X 0,Y 340.758,Z 303.039,A -85,B 0,C 180,E1 -14160.483,E2 -14160.483} C_VEL
LIN {X 0,Y 340.719,Z 303.043,A -85,B 0,C 180,E1 -14164.403,E2 -14164.403} C_VEL
LIN {X 0,Y 340.704,Z 303.044,A -85,B 0,C 180,E1 -14168.384,E2 -14168.384} C_VEL
LIN {X 0,Y 340.691,Z 303.048,A -85,B 0,C 180,E1 -14172.044,E2 -14172.044} C_VEL
LIN {X 0,Y 340.646,Z 303.05,A -85,B 0,C 180,E1 -14176.226,E2 -14176.226} C_VEL
LIN {X 0,Y 340.664,Z 303.047,A -85,B 0,C 180,E1 -14178.687,E2 -14178.687} C_VEL
LIN {X 0,Y 340.712,Z 303.046,A -85,B 0,C 180,E1 -14181.77,E2 -14181.77} C_VEL
LIN {X 0,Y 340.716,Z 303.044,A -85,B 0,C 180,E1 -14185.595,E2 -14185.595} C_VEL
LIN {X 0,Y 340.686,Z 303.044,A -85,B 0,C 180,E1 -14188.954,E2 -14188.954} C_VEL
LIN {X 0,Y 340.703,Z 303.044,A -85,B 0,C 180,E1 -14193.011,E2 -14193.011} C_VEL
LIN {X 0,Y 340.697,Z 303.044,A -85,B 0,C 180,E1 -14196.925,E2 -14196.925} C_VEL
LIN {X 0,Y 340.727,Z 303.037,A -85,B 0,C 180,E1 -14200.73,E2 -14200.73} C_VEL
LIN {X 0,Y 340.808,Z 303.026,A -85,B 0,C 180,E1 -14204.45,E2 -14204.45} C_VEL
LIN {X 0,Y 340.84,Z 303.025,A -85,B 0,C 180,E1 -14208.1,E2 -14208.1} C_VEL
LIN {X 0,Y 340.971,Z 303.007,A -85,B 0,C 180,E1 -14211.704,E2 -14211.704} C_VEL
LIN {X 0,Y 341,Z 302.998,A -85,B 0,C 180,E1 -14214.085,E2 -14214.085} C_VEL
LIN {X 0,Y 341.118,Z 302.991,A -85,B 0,C 180,E1 -14217.638,E2 -14217.638} C_VEL
LIN {X 0,Y 341.099,Z 302.998,A -85,B 0,C 180,E1 -14221.181,E2 -14221.181} C_VEL
LIN {X 0,Y 341.113,Z 302.991,A -85,B 0,C 180,E1 -14222.362,E2 -14222.362} C_VEL
LIN {X 0,Y 340.99,Z 303.011,A -85,B 0,C 180,E1 -14227.104,E2 -14227.104} C_VEL
LIN {X 0,Y 340.838,Z 303.027,A -85,B 0,C 180,E1 -14230.695,E2 -14230.695} C_VEL
LIN {X 0,Y 340.855,Z 303.024,A -85,B 0,C 180,E1 -14234.325,E2 -14234.325} C_VEL
LIN {X 0,Y 340.777,Z 303.033,A -85,B 0,C 180,E1 -14238.441,E2 -14238.441} C_VEL
LIN {X 0,Y 340.71,Z 303.041,A -85,B 0,C 180,E1 -14241.842,E2 -14241.842} C_VEL
LIN {X 0,Y 340.737,Z 303.036,A -85,B 0,C 180,E1 -14245.667,E2 -14245.667} C_VEL
LIN {X 0,Y 340.724,Z 303.039,A -85,B 0,C 180,E1 -14249.673,E2 -14249.673} C_VEL
LIN {X 0,Y 340.686,Z 303.044,A -85,B 0,C 180,E1 -14253.848,E2 -14253.848} C_VEL
LIN {X 0,Y 340.698,Z 303.045,A -85,B 0,C 180,E1 -14256.743,E2 -14256.743} C_VEL
LIN {X 0,Y 340.681,Z 303.048,A -85,B 0,C 180,E1 -14260.248,E2 -14260.248} C_VEL
LIN {X 0,Y 340.646,Z 303.049,A -85,B 0,C 180,E1 -14263.774,E2 -14263.774} C_VEL
LIN {X 0,Y 340.694,Z 303.044,A -85,B 0,C 180,E1 -14267.956,E2 -14267.956} C_VEL
LIN {X 0,Y 340.729,Z 303.039,A -85,B 0,C 180,E1 -14271.774,E2 -14271.774} C_VEL
LIN {X 0,Y 340.72,Z 303.041,A -85,B 0,C 180,E1 -14275.597,E2 -14275.597} C_VEL
LIN {X 0,Y 340.695,Z 303.043,A -85,B 0,C 180,E1 -14278.957,E2 -14278.957} C_VEL
LIN {X 0,Y 340.802,Z 303.03,A -85,B 0,C 180,E1 -14283.021,E2 -14283.021} C_VEL
LIN {X 0,Y 340.747,Z 303.041,A -85,B 0,C 180,E1 -14286.314,E2 -14286.314} C_VEL
LIN {X 0,Y 342.453,Z 307.393,A -85,B 0,C 180,E1 -14286.555,E2 -14286.555} C_VEL
LIN {X 0,Y 350.084,Z 324.968,A -85,B 0,C 180,E1 -14287.487,E2 -14287.487} C_VEL
LIN {X 0,Y 350.812,Z 331.853,A -85,B 0,C 180,E1 -14287.687,E2 -14287.687} C_VEL
LIN {X 0,Y 349.138,Z 414.857,A -85,B 0,C 180,E1 -14289.414,E2 -14289.414} C_VEL
LIN {X 0,Y 348.664,Z 428.244,A -85,B 0,C 180,E1 -14289.923,E2 -14289.923} C_VEL
LIN {X 0,Y 347.805,Z 441.307,A -85,B 0,C 180,E1 -14290.679,E2 -14290.679} C_VEL
LIN {X 0,Y 346.87,Z 452.435,A -85,B 0,C 180,E1 -14291.545,E2 -14291.545} C_VEL
LIN {X 0,Y 345.808,Z 463.277,A -85,B 0,C 180,E1 -14292.627,E2 -14292.627} C_VEL
LIN {X 0,Y 344.687,Z 474.238,A -85,B 0,C 180,E1 -14294.024,E2 -14294.024} C_VEL
LIN {X 0,Y 343.455,Z 483.538,A -85,B 0,C 180,E1 -14295.484,E2 -14295.484} C_VEL
LIN {X 0,Y 342.51,Z 491.15,A -85,B 0,C 180,E1 -14296.957,E2 -14296.957} C_VEL
LIN {X 0,Y 341.539,Z 498.575,A -85,B 0,C 180,E1 -14298.728,E2 -14298.728} C_VEL
LIN {X 0,Y 340.675,Z 504.539,A -85,B 0,C 180,E1 -14300.502,E2 -14300.502} C_VEL
LIN {X 0,Y 340.151,Z 509.247,A -85,B 0,C 180,E1 -14302.284,E2 -14302.284} C_VEL
LIN {X 0,Y 339.73,Z 512.845,A -85,B 0,C 180,E1 -14304.064,E2 -14304.064} C_VEL
LIN {X 0,Y 339.493,Z 514.7,A -85,B 0,C 180,E1 -14305.251,E2 -14305.251} C_VEL
LIN {X 0,Y 339.355,Z 516.115,A -85,B 0,C 180,E1 -14306.439,E2 -14306.439} C_VEL
LIN {X 0,Y 339.229,Z 517.717,A -85,B 0,C 180,E1 -14308.814,E2 -14308.814} C_VEL
LIN {X 0,Y 339.228,Z 517.95,A -85,B 0,C 180,E1 -14310.001,E2 -14310.001} C_VEL
LIN {X 0,Y 339.229,Z 517.758,A -85,B 0,C 180,E1 -14311.188,E2 -14311.188} C_VEL
LIN {X 0,Y 339.352,Z 516.211,A -85,B 0,C 180,E1 -14313.563,E2 -14313.563} C_VEL
LIN {X 0,Y 339.489,Z 514.85,A -85,B 0,C 180,E1 -14314.751,E2 -14314.751} C_VEL
LIN {X 0,Y 339.874,Z 511.812,A -85,B 0,C 180,E1 -14316.62,E2 -14316.62} C_VEL
LIN {X 0,Y 340.231,Z 508.094,A -85,B 0,C 180,E1 -14318.315,E2 -14318.315} C_VEL
LIN {X 0,Y 340.897,Z 503.05,A -85,B 0,C 180,E1 -14320.094,E2 -14320.094} C_VEL
LIN {X 0,Y 341.753,Z 496.688,A -85,B 0,C 180,E1 -14321.868,E2 -14321.868} C_VEL
LIN {X 0,Y 342.764,Z 488.771,A -85,B 0,C 180,E1 -14323.64,E2 -14323.64} C_VEL
LIN {X 0,Y 343.951,Z 480.662,A -85,B 0,C 180,E1 -14325.102,E2 -14325.102} C_VEL
LIN {X 0,Y 345.149,Z 470.703,A -85,B 0,C 180,E1 -14326.564,E2 -14326.564} C_VEL
LIN {X 0,Y 346.227,Z 459.512,A -85,B 0,C 180,E1 -14327.881,E2 -14327.881} C_VEL
LIN {X 0,Y 347.268,Z 448.507,A -85,B 0,C 180,E1 -14328.894,E2 -14328.894} C_VEL
LIN {X 0,Y 348.212,Z 436.07,A -85,B 0,C 180,E1 -14329.76,E2 -14329.76} C_VEL
LIN {X 0,Y 348.951,Z 423.068,A -85,B 0,C 180,E1 -14330.408,E2 -14330.408} C_VEL
LIN {X 0,Y 349.309,Z 410.342,A -85,B 0,C 180,E1 -14330.809,E2 -14330.809} C_VEL
LIN {X 0,Y 350.795,Z 329.759,A -85,B 0,C 180,E1 -14332.468,E2 -14332.468} C_VEL
LIN {X 0,Y 349.848,Z 324.336,A -85,B 0,C 180,E1 -14332.652,E2 -14332.652} C_VEL
LIN {X 0,Y 347.775,Z 319.399,A -85,B 0,C 180,E1 -14332.904,E2 -14332.904} C_VEL
LIN {X 0,Y 345.519,Z 316.326,A -85,B 0,C 180,E1 -14333.132,E2 -14333.132} C_VEL
LIN {X 0,Y 336.154,Z 308.969,A -85,B 0,C 180,E1 -14333.991,E2 -14333.991} C_VEL
LIN {X 0,Y 334.21,Z 305.82,A -85,B 0,C 180,E1 -14334.214,E2 -14334.214} C_VEL
LIN {X 0,Y 334.022,Z 305.215,A -85,B 0,C 180,E1 -14334.243,E2 -14334.243} C_VEL
LIN {X 0,Y 333.737,Z 303.911,A -85,B 0,C 180,E1 -14334.347,E2 -14334.347} C_VEL
LIN {X 0,Y 333.721,Z 303.916,A -85,B 0,C 180,E1 -14337.81,E2 -14337.81} C_VEL
LIN {X 0,Y 333.703,Z 303.916,A -85,B 0,C 180,E1 -14340.363,E2 -14340.363} C_VEL
LIN {X 0,Y 333.679,Z 303.918,A -85,B 0,C 180,E1 -14344.659,E2 -14344.659} C_VEL
LIN {X 0,Y 333.659,Z 303.926,A -85,B 0,C 180,E1 -14347.651,E2 -14347.651} C_VEL
LIN {X 0,Y 333.652,Z 303.922,A -85,B 0,C 180,E1 -14350.768,E2 -14350.768} C_VEL
LIN {X 0,Y 333.629,Z 303.921,A -85,B 0,C 180,E1 -14354.256,E2 -14354.256} C_VEL
LIN {X 0,Y 333.647,Z 303.922,A -85,B 0,C 180,E1 -14357.619,E2 -14357.619} C_VEL
LIN {X 0,Y 333.658,Z 303.925,A -85,B 0,C 180,E1 -14361.203,E2 -14361.203} C_VEL
LIN {X 0,Y 333.681,Z 303.916,A -85,B 0,C 180,E1 -14363.861,E2 -14363.861} C_VEL
LIN {X 0,Y 333.649,Z 303.922,A -85,B 0,C 180,E1 -14367.413,E2 -14367.413} C_VEL
LIN {X 0,Y 333.695,Z 303.92,A -85,B 0,C 180,E1 -14371.026,E2 -14371.026} C_VEL
LIN {X 0,Y 333.74,Z 303.91,A -85,B 0,C 180,E1 -14373.754,E2 -14373.754} C_VEL
LIN {X 0,Y 333.747,Z 304.059,A -85,B 0,C 180,E1 -14377.073,E2 -14377.073} C_VEL
LIN {X 0,Y 334.416,Z 307.604,A -85,B 0,C 180,E1 -14378.146,E2 -14378.146} C_VEL
LIN {X 0,Y 338.533,Z 323.074,A -85,B 0,C 180,E1 -14378.792,E2 -14378.792} C_VEL
LIN {X 0,Y 340.258,Z 333.691,A -85,B 0,C 180,E1 -14379.183,E2 -14379.183} C_VEL
LIN {X 0,Y 337.829,Z 416.024,A -85,B 0,C 180,E1 -14381.621,E2 -14381.621} C_VEL
LIN {X 0,Y 337.36,Z 429.677,A -85,B 0,C 180,E1 -14382.261,E2 -14382.261} C_VEL
LIN {X 0,Y 336.679,Z 441.272,A -85,B 0,C 180,E1 -14383.008,E2 -14383.008} C_VEL
LIN {X 0,Y 336.016,Z 453.769,A -85,B 0,C 180,E1 -14384.067,E2 -14384.067} C_VEL
LIN {X 0,Y 335.374,Z 465.246,A -85,B 0,C 180,E1 -14385.292,E2 -14385.292} C_VEL
LIN {X 0,Y 334.58,Z 475.448,A -85,B 0,C 180,E1 -14386.64,E2 -14386.64} C_VEL
LIN {X 0,Y 333.838,Z 484.828,A -85,B 0,C 180,E1 -14388.155,E2 -14388.155} C_VEL
LIN {X 0,Y 333.324,Z 492.607,A -85,B 0,C 180,E1 -14389.676,E2 -14389.676} C_VEL
LIN {X 0,Y 332.827,Z 500.252,A -85,B 0,C 180,E1 -14391.5,E2 -14391.5} C_VEL
LIN {X 0,Y 332.483,Z 506.712,A -85,B 0,C 180,E1 -14393.461,E2 -14393.461} C_VEL
LIN {X 0,Y 332.303,Z 511.078,A -85,B 0,C 180,E1 -14395.147,E2 -14395.147} C_VEL
LIN {X 0,Y 332.134,Z 514.676,A -85,B 0,C 180,E1 -14396.968,E2 -14396.968} C_VEL
LIN {X 0,Y 332.069,Z 517.21,A -85,B 0,C 180,E1 -14398.787,E2 -14398.787} C_VEL
LIN {X 0,Y 332.099,Z 518.34,A -85,B 0,C 180,E1 -14400,E2 -14400} C_VEL
LIN {X 0,Y 332.193,Z 519.045,A -85,B 0,C 180,E1 -14401.212,E2 -14401.212} C_VEL
LIN {X 0,Y 332.345,Z 519.275,A -85,B 0,C 180,E1 -14402.424,E2 -14402.424} C_VEL
LIN {X 0,Y 332.549,Z 519.081,A -85,B 0,C 180,E1 -14403.635,E2 -14403.635} C_VEL
LIN {X 0,Y 332.65,Z 518.486,A -85,B 0,C 180,E1 -14404.848,E2 -14404.848} C_VEL
LIN {X 0,Y 332.822,Z 517.455,A -85,B 0,C 180,E1 -14406.061,E2 -14406.061} C_VEL
LIN {X 0,Y 333.625,Z 514.7,A -85,B 0,C 180,E1 -14408.07,E2 -14408.07} C_VEL
LIN {X 0,Y 334.657,Z 510.183,A -85,B 0,C 180,E1 -14410.283,E2 -14410.283} C_VEL
LIN {X 0,Y 335.731,Z 505.219,A -85,B 0,C 180,E1 -14412.083,E2 -14412.083} C_VEL
LIN {X 0,Y 337.004,Z 498.958,A -85,B 0,C 180,E1 -14413.876,E2 -14413.876} C_VEL
LIN {X 0,Y 338.507,Z 491.134,A -85,B 0,C 180,E1 -14415.658,E2 -14415.658} C_VEL
LIN {X 0,Y 340.445,Z 481.447,A -85,B 0,C 180,E1 -14417.417,E2 -14417.417} C_VEL
LIN {X 0,Y 342.435,Z 470.226,A -85,B 0,C 180,E1 -14419.025,E2 -14419.025} C_VEL
LIN {X 0,Y 344.22,Z 459.007,A -85,B 0,C 180,E1 -14420.31,E2 -14420.31} C_VEL
LIN {X 0,Y 345.98,Z 446.331,A -85,B 0,C 180,E1 -14421.447,E2 -14421.447} C_VEL
LIN {X 0,Y 347.308,Z 434.166,A -85,B 0,C 180,E1 -14422.298,E2 -14422.298} C_VEL
LIN {X 0,Y 348.622,Z 419.592,A -85,B 0,C 180,E1 -14423.03,E2 -14423.03} C_VEL
LIN {X 0,Y 354.34,Z 345.458,A -85,B 0,C 180,E1 -14425.619,E2 -14425.619} C_VEL
LIN {X 0,Y 349.888,Z 336.356,A -85,B 0,C 180,E1 -14426.81,E2 -14426.81} C_VEL
LIN {X 0,Y 345.465,Z 328.754,A -85,B 0,C 180,E1 -14428.046,E2 -14428.046} C_VEL
LIN {X 0,Y 342.808,Z 324.593,A -85,B 0,C 180,E1 -14428.837,E2 -14428.837} C_VEL
LIN {X 0,Y 340.266,Z 320.792,A -85,B 0,C 180,E1 -14429.634,E2 -14429.634} C_VEL
LIN {X 0,Y 337.703,Z 317.155,A -85,B 0,C 180,E1 -14430.488,E2 -14430.488} C_VEL
LIN {X 0,Y 337.427,Z 316.526,A -85,B 0,C 180,E1 -14430.684,E2 -14430.684} C_VEL
LIN {X 0,Y 336.561,Z 313.293,A -85,B 0,C 180,E1 -14433.354,E2 -14433.354} C_VEL
LIN {X 0,Y 335.854,Z 311.016,A -85,B 0,C 180,E1 -14435.868,E2 -14435.868} C_VEL
LIN {X 0,Y 335.358,Z 309.14,A -85,B 0,C 180,E1 -14439.158,E2 -14439.158} C_VEL
LIN {X 0,Y 335.172,Z 308.759,A -85,B 0,C 180,E1 -14442.785,E2 -14442.785} C_VEL
LIN {X 0,Y 335.518,Z 309.467,A -85,B 0,C 180,E1 -14445.413,E2 -14445.413} C_VEL
LIN {X 0,Y 336.178,Z 311.865,A -85,B 0,C 180,E1 -14448.816,E2 -14448.816} C_VEL
LIN {X 0,Y 337.05,Z 314.518,A -85,B 0,C 180,E1 -14451.277,E2 -14451.277} C_VEL
LIN {X 0,Y 337.802,Z 316.679,A -85,B 0,C 180,E1 -14452.889,E2 -14452.889} C_VEL
LIN {X 0,Y 339.206,Z 321.951,A -85,B 0,C 180,E1 -14455.984,E2 -14455.984} C_VEL
LIN {X 0,Y 340.751,Z 328.279,A -85,B 0,C 180,E1 -14458.96,E2 -14458.96} C_VEL
LIN {X 0,Y 341.483,Z 331.932,A -85,B 0,C 180,E1 -14460.367,E2 -14460.367} C_VEL
LIN {X 0,Y 344.094,Z 337.028,A -85,B 0,C 180,E1 -14461.199,E2 -14461.199} C_VEL
LIN {X 0,Y 346.481,Z 342.631,A -85,B 0,C 180,E1 -14461.96,E2 -14461.96} C_VEL
LIN {X 0,Y 349.172,Z 354.723,A -85,B 0,C 180,E1 -14463.062,E2 -14463.062} C_VEL
LIN {X 0,Y 351.331,Z 367.923,A -85,B 0,C 180,E1 -14464.056,E2 -14464.056} C_VEL
LIN {X 0,Y 352.411,Z 379.005,A -85,B 0,C 180,E1 -14464.734,E2 -14464.734} C_VEL
LIN {X 0,Y 347.347,Z 446.742,A -85,B 0,C 180,E1 -14467.076,E2 -14467.076} C_VEL
LIN {X 0,Y 345.868,Z 460.149,A -85,B 0,C 180,E1 -14467.761,E2 -14467.761} C_VEL
LIN {X 0,Y 344.177,Z 472.38,A -85,B 0,C 180,E1 -14468.591,E2 -14468.591} C_VEL
LIN {X 0,Y 342.416,Z 483.761,A -85,B 0,C 180,E1 -14469.578,E2 -14469.578} C_VEL
LIN {X 0,Y 340.481,Z 495.539,A -85,B 0,C 180,E1 -14470.871,E2 -14470.871} C_VEL
LIN {X 0,Y 338.763,Z 505.247,A -85,B 0,C 180,E1 -14472.18,E2 -14472.18} C_VEL
LIN {X 0,Y 336.766,Z 515.475,A -85,B 0,C 180,E1 -14473.857,E2 -14473.857} C_VEL
LIN {X 0,Y 335.304,Z 524.496,A -85,B 0,C 180,E1 -14475.741,E2 -14475.741} C_VEL
LIN {X 0,Y 334.013,Z 531.526,A -85,B 0,C 180,E1 -14477.544,E2 -14477.544} C_VEL
LIN {X 0,Y 333.012,Z 537.993,A -85,B 0,C 180,E1 -14479.665,E2 -14479.665} C_VEL
LIN {X 0,Y 332.462,Z 542.26,A -85,B 0,C 180,E1 -14481.489,E2 -14481.489} C_VEL
LIN {X 0,Y 332.183,Z 544.491,A -85,B 0,C 180,E1 -14482.706,E2 -14482.706} C_VEL
LIN {X 0,Y 332.032,Z 546.598,A -85,B 0,C 180,E1 -14484.174,E2 -14484.174} C_VEL
LIN {X 0,Y 332.013,Z 548.496,A -85,B 0,C 180,E1 -14486.358,E2 -14486.358} C_VEL
LIN {X 0,Y 331.981,Z 548.951,A -85,B 0,C 180,E1 -14487.572,E2 -14487.572} C_VEL
LIN {X 0,Y 332.099,Z 548.982,A -85,B 0,C 180,E1 -14488.786,E2 -14488.786} C_VEL
LIN {X 0,Y 332.239,Z 548.53,A -85,B 0,C 180,E1 -14489.999,E2 -14489.999} C_VEL
LIN {X 0,Y 332.092,Z 547.09,A -85,B 0,C 180,E1 -14492.425,E2 -14492.425} C_VEL
LIN {X 0,Y 332.064,Z 546.071,A -85,B 0,C 180,E1 -14493.639,E2 -14493.639} C_VEL
LIN {X 0,Y 332.095,Z 542.964,A -85,B 0,C 180,E1 -14495.931,E2 -14495.931} C_VEL
LIN {X 0,Y 332.263,Z 539.011,A -85,B 0,C 180,E1 -14497.901,E2 -14497.901} C_VEL
LIN {X 0,Y 332.606,Z 534.166,A -85,B 0,C 180,E1 -14499.731,E2 -14499.731} C_VEL
LIN {X 0,Y 333.189,Z 528.039,A -85,B 0,C 180,E1 -14501.558,E2 -14501.558} C_VEL
LIN {X 0,Y 334.19,Z 520.42,A -85,B 0,C 180,E1 -14503.374,E2 -14503.374} C_VEL
LIN {X 0,Y 335.308,Z 511.772,A -85,B 0,C 180,E1 -14505.021,E2 -14505.021} C_VEL
LIN {X 0,Y 336.407,Z 501.958,A -85,B 0,C 180,E1 -14506.536,E2 -14506.536} C_VEL
LIN {X 0,Y 337.536,Z 492.399,A -85,B 0,C 180,E1 -14507.728,E2 -14507.728} C_VEL
LIN {X 0,Y 338.761,Z 482.114,A -85,B 0,C 180,E1 -14508.756,E2 -14508.756} C_VEL
LIN {X 0,Y 339.876,Z 469.751,A -85,B 0,C 180,E1 -14509.712,E2 -14509.712} C_VEL
LIN {X 0,Y 340.882,Z 456.757,A -85,B 0,C 180,E1 -14510.437,E2 -14510.437} C_VEL
LIN {X 0,Y 341.545,Z 445.097,A -85,B 0,C 180,E1 -14510.868,E2 -14510.868} C_VEL
LIN {X 0,Y 342.854,Z 375.979,A -85,B 0,C 180,E1 -14512.332,E2 -14512.332} C_VEL
LIN {X 0,Y 338.333,Z 343.131,A -85,B 0,C 180,E1 -14513.381,E2 -14513.381} C_VEL
LIN {X 0,Y 336.46,Z 330.88,A -85,B 0,C 180,E1 -14513.799,E2 -14513.799} C_VEL
LIN {X 0,Y 337.278,Z 323.298,A -85,B 0,C 180,E1 -14515.617,E2 -14515.617} C_VEL
LIN {X 0,Y 336.718,Z 318.765,A -85,B 0,C 180,E1 -14516.756,E2 -14516.756} C_VEL
LIN {X 0,Y 333.927,Z 305.013,A -85,B 0,C 180,E1 -14520.355,E2 -14520.355} C_VEL
LIN {X 0,Y 333.704,Z 303.916,A -85,B 0,C 180,E1 -14520.709,E2 -14520.709} C_VEL
LIN {X 0,Y 333.682,Z 303.918,A -85,B 0,C 180,E1 -14524.773,E2 -14524.773} C_VEL
LIN {X 0,Y 333.647,Z 303.923,A -85,B 0,C 180,E1 -14527.65,E2 -14527.65} C_VEL
LIN {X 0,Y 333.64,Z 303.922,A -85,B 0,C 180,E1 -14530.766,E2 -14530.766} C_VEL
LIN {X 0,Y 333.588,Z 303.931,A -85,B 0,C 180,E1 -14534.249,E2 -14534.249} C_VEL
LIN {X 0,Y 333.632,Z 303.925,A -85,B 0,C 180,E1 -14537.617,E2 -14537.617} C_VEL
LIN {X 0,Y 333.609,Z 303.925,A -85,B 0,C 180,E1 -14541.209,E2 -14541.209} C_VEL
LIN {X 0,Y 333.668,Z 303.921,A -85,B 0,C 180,E1 -14543.86,E2 -14543.86} C_VEL
LIN {X 0,Y 333.636,Z 303.926,A -85,B 0,C 180,E1 -14547.412,E2 -14547.412} C_VEL
LIN {X 0,Y 333.623,Z 303.925,A -85,B 0,C 180,E1 -14551.02,E2 -14551.02} C_VEL
LIN {X 0,Y 333.651,Z 303.92,A -85,B 0,C 180,E1 -14554.921,E2 -14554.921} C_VEL
LIN {X 0,Y 333.656,Z 303.922,A -85,B 0,C 180,E1 -14559.018,E2 -14559.018} C_VEL
LIN {X 0,Y 333.732,Z 303.907,A -85,B 0,C 180,E1 -14561.586,E2 -14561.586} C_VEL
LIN {X 0,Y 333.8,Z 303.905,A -85,B 0,C 180,E1 -14565.576,E2 -14565.576} C_VEL
LIN {X 0,Y 333.808,Z 303.905,A -85,B 0,C 180,E1 -14569.077,E2 -14569.077} C_VEL
LIN {X 0,Y 333.944,Z 303.881,A -85,B 0,C 180,E1 -14572.746,E2 -14572.746} C_VEL
LIN {X 0,Y 333.771,Z 303.901,A -85,B 0,C 180,E1 -14575.169,E2 -14575.169} C_VEL
LIN {X 0,Y 334.059,Z 303.871,A -85,B 0,C 180,E1 -14577.589,E2 -14577.589} C_VEL
LIN {X 0,Y 334.068,Z 303.873,A -85,B 0,C 180,E1 -14581.206,E2 -14581.206} C_VEL
LIN {X 0,Y 334.054,Z 303.87,A -85,B 0,C 180,E1 -14582.412,E2 -14582.412} C_VEL
LIN {X 0,Y 333.944,Z 303.883,A -85,B 0,C 180,E1 -14586.583,E2 -14586.583} C_VEL
LIN {X 0,Y 333.811,Z 303.899,A -85,B 0,C 180,E1 -14589.697,E2 -14589.697} C_VEL
LIN {X 0,Y 333.788,Z 303.905,A -85,B 0,C 180,E1 -14593.392,E2 -14593.392} C_VEL
LIN {X 0,Y 333.711,Z 303.914,A -85,B 0,C 180,E1 -14597.148,E2 -14597.148} C_VEL
LIN {X 0,Y 333.677,Z 303.917,A -85,B 0,C 180,E1 -14599.694,E2 -14599.694} C_VEL
LIN {X 0,Y 333.66,Z 303.918,A -85,B 0,C 180,E1 -14603.591,E2 -14603.591} C_VEL
LIN {X 0,Y 333.668,Z 303.918,A -85,B 0,C 180,E1 -14606.252,E2 -14606.252} C_VEL
LIN {X 0,Y 333.653,Z 303.923,A -85,B 0,C 180,E1 -14610.367,E2 -14610.367} C_VEL
LIN {X 0,Y 333.63,Z 303.924,A -85,B 0,C 180,E1 -14613.209,E2 -14613.209} C_VEL
LIN {X 0,Y 333.669,Z 303.921,A -85,B 0,C 180,E1 -14616.14,E2 -14616.14} C_VEL
LIN {X 0,Y 333.64,Z 303.922,A -85,B 0,C 180,E1 -14619.194,E2 -14619.194} C_VEL
LIN {X 0,Y 333.627,Z 303.927,A -85,B 0,C 180,E1 -14622.501,E2 -14622.501} C_VEL
LIN {X 0,Y 333.591,Z 303.93,A -85,B 0,C 180,E1 -14625.956,E2 -14625.956} C_VEL
LIN {X 0,Y 333.643,Z 303.922,A -85,B 0,C 180,E1 -14629.317,E2 -14629.317} C_VEL
LIN {X 0,Y 333.661,Z 303.916,A -85,B 0,C 180,E1 -14633.169,E2 -14633.169} C_VEL
LIN {X 0,Y 333.671,Z 303.919,A -85,B 0,C 180,E1 -14635.343,E2 -14635.343} C_VEL
LIN {X 0,Y 333.688,Z 303.917,A -85,B 0,C 180,E1 -14639.639,E2 -14639.639} C_VEL
LIN {X 0,Y 333.738,Z 303.913,A -85,B 0,C 180,E1 -14642.402,E2 -14642.402} C_VEL
LIN {X 0,Y 333.712,Z 303.914,A -85,B 0,C 180,E1 -14645.814,E2 -14645.814} C_VEL
LIN {X 0,Y 334.813,Z 306.939,A -85,B 0,C 180,E1 -14645.97,E2 -14645.97} C_VEL
LIN {X 0,Y 343.763,Z 327.29,A -85,B 0,C 180,E1 -14647.096,E2 -14647.096} C_VEL
LIN {X 0,Y 344.252,Z 332.531,A -85,B 0,C 180,E1 -14647.248,E2 -14647.248} C_VEL
LIN {X 0,Y 342.522,Z 415.115,A -85,B 0,C 180,E1 -14648.998,E2 -14648.998} C_VEL
LIN {X 0,Y 342.073,Z 427.77,A -85,B 0,C 180,E1 -14649.48,E2 -14649.48} C_VEL
LIN {X 0,Y 341.188,Z 440.538,A -85,B 0,C 180,E1 -14650.21,E2 -14650.21} C_VEL
LIN {X 0,Y 340.167,Z 452.74,A -85,B 0,C 180,E1 -14651.168,E2 -14651.168} C_VEL
LIN {X 0,Y 339.029,Z 463.8,A -85,B 0,C 180,E1 -14652.295,E2 -14652.295} C_VEL
LIN {X 0,Y 337.888,Z 474.55,A -85,B 0,C 180,E1 -14653.694,E2 -14653.694} C_VEL
LIN {X 0,Y 336.592,Z 483.852,A -85,B 0,C 180,E1 -14655.182,E2 -14655.182} C_VEL
LIN {X 0,Y 335.597,Z 491.466,A -85,B 0,C 180,E1 -14656.683,E2 -14656.683} C_VEL
LIN {X 0,Y 334.563,Z 498.892,A -85,B 0,C 180,E1 -14658.49,E2 -14658.49} C_VEL
LIN {X 0,Y 333.669,Z 504.856,A -85,B 0,C 180,E1 -14660.301,E2 -14660.301} C_VEL
LIN {X 0,Y 333.12,Z 509.563,A -85,B 0,C 180,E1 -14662.119,E2 -14662.119} C_VEL
LIN {X 0,Y 332.676,Z 513.163,A -85,B 0,C 180,E1 -14663.938,E2 -14663.938} C_VEL
LIN {X 0,Y 332.439,Z 515.017,A -85,B 0,C 180,E1 -14665.15,E2 -14665.15} C_VEL
LIN {X 0,Y 332.277,Z 516.432,A -85,B 0,C 180,E1 -14666.363,E2 -14666.363} C_VEL
LIN {X 0,Y 332.137,Z 518.034,A -85,B 0,C 180,E1 -14668.789,E2 -14668.789} C_VEL
LIN {X 0,Y 332.136,Z 518.266,A -85,B 0,C 180,E1 -14670.001,E2 -14670.001} C_VEL
LIN {X 0,Y 332.137,Z 518.075,A -85,B 0,C 180,E1 -14671.214,E2 -14671.214} C_VEL
LIN {X 0,Y 332.274,Z 516.527,A -85,B 0,C 180,E1 -14673.639,E2 -14673.639} C_VEL
LIN {X 0,Y 332.435,Z 515.165,A -85,B 0,C 180,E1 -14674.852,E2 -14674.852} C_VEL
LIN {X 0,Y 332.894,Z 511.388,A -85,B 0,C 180,E1 -14677.133,E2 -14677.133} C_VEL
LIN {X 0,Y 333.391,Z 506.843,A -85,B 0,C 180,E1 -14679.098,E2 -14679.098} C_VEL
LIN {X 0,Y 334.207,Z 501.4,A -85,B 0,C 180,E1 -14680.911,E2 -14680.911} C_VEL
LIN {X 0,Y 335.146,Z 494.572,A -85,B 0,C 180,E1 -14682.721,E2 -14682.721} C_VEL
LIN {X 0,Y 336.351,Z 486.01,A -85,B 0,C 180,E1 -14684.522,E2 -14684.522} C_VEL
LIN {X 0,Y 337.587,Z 477.235,A -85,B 0,C 180,E1 -14686.013,E2 -14686.013} C_VEL
LIN {X 0,Y 338.632,Z 467.94,A -85,B 0,C 180,E1 -14687.313,E2 -14687.313} C_VEL
LIN {X 0,Y 339.78,Z 456.908,A -85,B 0,C 180,E1 -14688.544,E2 -14688.544} C_VEL
LIN {X 0,Y 340.915,Z 445.024,A -85,B 0,C 180,E1 -14689.573,E2 -14689.573} C_VEL
LIN {X 0,Y 341.778,Z 432.57,A -85,B 0,C 180,E1 -14690.384,E2 -14690.384} C_VEL
LIN {X 0,Y 342.476,Z 419.366,A -85,B 0,C 180,E1 -14690.969,E2 -14690.969} C_VEL
LIN {X 0,Y 342.82,Z 405.341,A -85,B 0,C 180,E1 -14691.34,E2 -14691.34} C_VEL
LIN {X 0,Y 344.24,Z 330.635,A -85,B 0,C 180,E1 -14692.904,E2 -14692.904} C_VEL
LIN {X 0,Y 343.497,Z 326.589,A -85,B 0,C 180,E1 -14693.048,E2 -14693.048} C_VEL
LIN {X 0,Y 334.624,Z 306.594,A -85,B 0,C 180,E1 -14694.164,E2 -14694.164} C_VEL
LIN {X 0,Y 334.022,Z 305.215,A -85,B 0,C 180,E1 -14694.243,E2 -14694.243} C_VEL
LIN {X 0,Y 333.354,Z 304.205,A -85,B 0,C 180,E1 -14694.426,E2 -14694.426} C_VEL
LIN {X 0,Y 331.59,Z 304.177,A -85,B 0,C 180,E1 -14695.094,E2 -14695.094} C_VEL
LIN {X 0,Y 328.928,Z 304.662,A -85,B 0,C 180,E1 -14696.556,E2 -14696.556} C_VEL
LIN {X 0,Y 327.339,Z 305.05,A -85,B 0,C 180,E1 -14697.944,E2 -14697.944} C_VEL
LIN {X 0,Y 326.659,Z 304.795,A -85,B 0,C 180,E1 -14699.571,E2 -14699.571} C_VEL
LIN {X 0,Y 326.624,Z 304.798,A -85,B 0,C 180,E1 -14702.947,E2 -14702.947} C_VEL
LIN {X 0,Y 326.618,Z 304.803,A -85,B 0,C 180,E1 -14705.52,E2 -14705.52} C_VEL
LIN {X 0,Y 326.617,Z 304.802,A -85,B 0,C 180,E1 -14709.228,E2 -14709.228} C_VEL
LIN {X 0,Y 326.587,Z 304.805,A -85,B 0,C 180,E1 -14712.974,E2 -14712.974} C_VEL
LIN {X 0,Y 326.588,Z 304.795,A -85,B 0,C 180,E1 -14717.027,E2 -14717.027} C_VEL
LIN {X 0,Y 326.616,Z 304.8,A -85,B 0,C 180,E1 -14720.773,E2 -14720.773} C_VEL
LIN {X 0,Y 326.617,Z 304.796,A -85,B 0,C 180,E1 -14724.481,E2 -14724.481} C_VEL
LIN {X 0,Y 326.613,Z 304.798,A -85,B 0,C 180,E1 -14727.456,E2 -14727.456} C_VEL
LIN {X 0,Y 326.653,Z 304.791,A -85,B 0,C 180,E1 -14730.34,E2 -14730.34} C_VEL
LIN {X 0,Y 326.695,Z 304.79,A -85,B 0,C 180,E1 -14734.517,E2 -14734.517} C_VEL
LIN {X 0,Y 326.72,Z 304.892,A -85,B 0,C 180,E1 -14736.927,E2 -14736.927} C_VEL
LIN {X 0,Y 327.288,Z 308.034,A -85,B 0,C 180,E1 -14737.86,E2 -14737.86} C_VEL
LIN {X 0,Y 331.855,Z 325.36,A -85,B 0,C 180,E1 -14738.6,E2 -14738.6} C_VEL
LIN {X 0,Y 333.308,Z 334.818,A -85,B 0,C 180,E1 -14738.954,E2 -14738.954} C_VEL
LIN {X 0,Y 330.823,Z 416.513,A -85,B 0,C 180,E1 -14741.458,E2 -14741.458} C_VEL
LIN {X 0,Y 330.311,Z 430.055,A -85,B 0,C 180,E1 -14742.11,E2 -14742.11} C_VEL
LIN {X 0,Y 329.609,Z 442.622,A -85,B 0,C 180,E1 -14742.951,E2 -14742.951} C_VEL
LIN {X 0,Y 328.841,Z 456.141,A -85,B 0,C 180,E1 -14744.152,E2 -14744.152} C_VEL
LIN {X 0,Y 328.096,Z 467.319,A -85,B 0,C 180,E1 -14745.422,E2 -14745.422} C_VEL
LIN {X 0,Y 327.323,Z 477.288,A -85,B 0,C 180,E1 -14746.813,E2 -14746.813} C_VEL
LIN {X 0,Y 326.615,Z 487.273,A -85,B 0,C 180,E1 -14748.519,E2 -14748.519} C_VEL
LIN {X 0,Y 326.015,Z 495.996,A -85,B 0,C 180,E1 -14750.382,E2 -14750.382} C_VEL
LIN {X 0,Y 325.554,Z 503.037,A -85,B 0,C 180,E1 -14752.246,E2 -14752.246} C_VEL
LIN {X 0,Y 325.305,Z 507.767,A -85,B 0,C 180,E1 -14753.799,E2 -14753.799} C_VEL
LIN {X 0,Y 325.185,Z 512.301,A -85,B 0,C 180,E1 -14755.662,E2 -14755.662} C_VEL
LIN {X 0,Y 325.013,Z 515.676,A -85,B 0,C 180,E1 -14757.521,E2 -14757.521} C_VEL
LIN {X 0,Y 324.973,Z 517.343,A -85,B 0,C 180,E1 -14758.761,E2 -14758.761} C_VEL
LIN {X 0,Y 325.003,Z 518.539,A -85,B 0,C 180,E1 -14760,E2 -14760} C_VEL
LIN {X 0,Y 325.101,Z 519.321,A -85,B 0,C 180,E1 -14761.239,E2 -14761.239} C_VEL
LIN {X 0,Y 325.262,Z 519.674,A -85,B 0,C 180,E1 -14762.477,E2 -14762.477} C_VEL
LIN {X 0,Y 325.47,Z 519.555,A -85,B 0,C 180,E1 -14763.714,E2 -14763.714} C_VEL
LIN {X 0,Y 325.585,Z 519.031,A -85,B 0,C 180,E1 -14764.953,E2 -14764.953} C_VEL
LIN {X 0,Y 325.801,Z 518.096,A -85,B 0,C 180,E1 -14766.192,E2 -14766.192} C_VEL
LIN {X 0,Y 326.616,Z 515.621,A -85,B 0,C 180,E1 -14768.18,E2 -14768.18} C_VEL
LIN {X 0,Y 327.423,Z 512.515,A -85,B 0,C 180,E1 -14769.888,E2 -14769.888} C_VEL
LIN {X 0,Y 328.471,Z 508.125,A -85,B 0,C 180,E1 -14771.728,E2 -14771.728} C_VEL
LIN {X 0,Y 329.961,Z 501.42,A -85,B 0,C 180,E1 -14773.864,E2 -14773.864} C_VEL
LIN {X 0,Y 331.586,Z 494.143,A -85,B 0,C 180,E1 -14775.678,E2 -14775.678} C_VEL
LIN {X 0,Y 333.18,Z 486.749,A -85,B 0,C 180,E1 -14777.176,E2 -14777.176} C_VEL
LIN {X 0,Y 335.231,Z 476.778,A -85,B 0,C 180,E1 -14778.814,E2 -14778.814} C_VEL
LIN {X 0,Y 337.198,Z 466.235,A -85,B 0,C 180,E1 -14780.209,E2 -14780.209} C_VEL
LIN {X 0,Y 338.985,Z 454.803,A -85,B 0,C 180,E1 -14781.433,E2 -14781.433} C_VEL
LIN {X 0,Y 340.91,Z 440.918,A -85,B 0,C 180,E1 -14782.579,E2 -14782.579} C_VEL
LIN {X 0,Y 342.283,Z 428.173,A -85,B 0,C 180,E1 -14783.362,E2 -14783.362} C_VEL
LIN {X 0,Y 343.506,Z 413.652,A -85,B 0,C 180,E1 -14783.994,E2 -14783.994} C_VEL
LIN {X 0,Y 349.092,Z 348.495,A -85,B 0,C 180,E1 -14786.312,E2 -14786.312} C_VEL
LIN {X 0,Y 345.675,Z 341.194,A -85,B 0,C 180,E1 -14787.304,E2 -14787.304} C_VEL
LIN {X 0,Y 341.515,Z 333.889,A -85,B 0,C 180,E1 -14788.537,E2 -14788.537} C_VEL
LIN {X 0,Y 338.954,Z 329.803,A -85,B 0,C 180,E1 -14789.345,E2 -14789.345} C_VEL
LIN {X 0,Y 336.707,Z 326.366,A -85,B 0,C 180,E1 -14790.097,E2 -14790.097} C_VEL
LIN {X 0,Y 333.637,Z 322.043,A -85,B 0,C 180,E1 -14791.192,E2 -14791.192} C_VEL
LIN {X 0,Y 330.897,Z 318.349,A -85,B 0,C 180,E1 -14792.259,E2 -14792.259} C_VEL
LIN {X 0,Y 330.601,Z 317.682,A -85,B 0,C 180,E1 -14792.464,E2 -14792.464} C_VEL
LIN {X 0,Y 329.708,Z 314.509,A -85,B 0,C 180,E1 -14795.902,E2 -14795.902} C_VEL
LIN {X 0,Y 329.343,Z 313.155,A -85,B 0,C 180,E1 -14798.232,E2 -14798.232} C_VEL
LIN {X 0,Y 329.061,Z 312.378,A -85,B 0,C 180,E1 -14801.623,E2 -14801.623} C_VEL
LIN {X 0,Y 329.389,Z 313.057,A -85,B 0,C 180,E1 -14805.241,E2 -14805.241} C_VEL
LIN {X 0,Y 329.906,Z 314.97,A -85,B 0,C 180,E1 -14808.211,E2 -14808.211} C_VEL
LIN {X 0,Y 330.574,Z 317.04,A -85,B 0,C 180,E1 -14810.371,E2 -14810.371} C_VEL
LIN {X 0,Y 331.592,Z 320.092,A -85,B 0,C 180,E1 -14812.839,E2 -14812.839} C_VEL
LIN {X 0,Y 332.891,Z 325.094,A -85,B 0,C 180,E1 -14815.855,E2 -14815.855} C_VEL
LIN {X 0,Y 334.282,Z 330.921,A -85,B 0,C 180,E1 -14818.642,E2 -14818.642} C_VEL
LIN {X 0,Y 336.987,Z 336.127,A -85,B 0,C 180,E1 -14819.644,E2 -14819.644} C_VEL
LIN {X 0,Y 340.552,Z 343.138,A -85,B 0,C 180,E1 -14820.848,E2 -14820.848} C_VEL
LIN {X 0,Y 342.052,Z 347.043,A -85,B 0,C 180,E1 -14821.375,E2 -14821.375} C_VEL
LIN {X 0,Y 344.491,Z 359.096,A -85,B 0,C 180,E1 -14822.495,E2 -14822.495} C_VEL
LIN {X 0,Y 346.442,Z 372.565,A -85,B 0,C 180,E1 -14823.525,E2 -14823.525} C_VEL
LIN {X 0,Y 346.982,Z 381.229,A -85,B 0,C 180,E1 -14824.038,E2 -14824.038} C_VEL
LIN {X 0,Y 341.698,Z 446.213,A -85,B 0,C 180,E1 -14826.354,E2 -14826.354} C_VEL
LIN {X 0,Y 340.118,Z 459.511,A -85,B 0,C 180,E1 -14827.043,E2 -14827.043} C_VEL
LIN {X 0,Y 338.296,Z 471.674,A -85,B 0,C 180,E1 -14827.879,E2 -14827.879} C_VEL
LIN {X 0,Y 336.182,Z 484.476,A -85,B 0,C 180,E1 -14829.021,E2 -14829.021} C_VEL
LIN {X 0,Y 334.105,Z 495.977,A -85,B 0,C 180,E1 -14830.331,E2 -14830.331} C_VEL
LIN {X 0,Y 332.107,Z 506.494,A -85,B 0,C 180,E1 -14831.811,E2 -14831.811} C_VEL
LIN {X 0,Y 330.03,Z 516.29,A -85,B 0,C 180,E1 -14833.511,E2 -14833.511} C_VEL
LIN {X 0,Y 328.453,Z 525.125,A -85,B 0,C 180,E1 -14835.437,E2 -14835.437} C_VEL
LIN {X 0,Y 327.099,Z 531.93,A -85,B 0,C 180,E1 -14837.276,E2 -14837.276} C_VEL
LIN {X 0,Y 326.012,Z 538.182,A -85,B 0,C 180,E1 -14839.44,E2 -14839.44} C_VEL
LIN {X 0,Y 325.427,Z 542.3,A -85,B 0,C 180,E1 -14841.304,E2 -14841.304} C_VEL
LIN {X 0,Y 325.137,Z 544.468,A -85,B 0,C 180,E1 -14842.547,E2 -14842.547} C_VEL
LIN {X 0,Y 324.926,Z 546.656,A -85,B 0,C 180,E1 -14844.246,E2 -14844.246} C_VEL
LIN {X 0,Y 324.938,Z 548.219,A -85,B 0,C 180,E1 -14846.278,E2 -14846.278} C_VEL
LIN {X 0,Y 324.897,Z 548.612,A -85,B 0,C 180,E1 -14847.519,E2 -14847.519} C_VEL
LIN {X 0,Y 325.008,Z 548.533,A -85,B 0,C 180,E1 -14848.76,E2 -14848.76} C_VEL
LIN {X 0,Y 325.132,Z 547.405,A -85,B 0,C 180,E1 -14851.237,E2 -14851.237} C_VEL
LIN {X 0,Y 324.987,Z 545.754,A -85,B 0,C 180,E1 -14853.718,E2 -14853.718} C_VEL
LIN {X 0,Y 325.001,Z 542.952,A -85,B 0,C 180,E1 -14855.883,E2 -14855.883} C_VEL
LIN {X 0,Y 325.193,Z 538.692,A -85,B 0,C 180,E1 -14858.074,E2 -14858.074} C_VEL
LIN {X 0,Y 325.559,Z 533.847,A -85,B 0,C 180,E1 -14859.944,E2 -14859.944} C_VEL
LIN {X 0,Y 326.178,Z 527.72,A -85,B 0,C 180,E1 -14861.81,E2 -14861.81} C_VEL
LIN {X 0,Y 327.237,Z 520.103,A -85,B 0,C 180,E1 -14863.664,E2 -14863.664} C_VEL
LIN {X 0,Y 328.333,Z 512.203,A -85,B 0,C 180,E1 -14865.214,E2 -14865.214} C_VEL
LIN {X 0,Y 329.432,Z 502.71,A -85,B 0,C 180,E1 -14866.737,E2 -14866.737} C_VEL
LIN {X 0,Y 330.761,Z 492.09,A -85,B 0,C 180,E1 -14868.103,E2 -14868.103} C_VEL
LIN {X 0,Y 332.007,Z 481.807,A -85,B 0,C 180,E1 -14869.153,E2 -14869.153} C_VEL
LIN {X 0,Y 333.208,Z 469.453,A -85,B 0,C 180,E1 -14870.123,E2 -14870.123} C_VEL
LIN {X 0,Y 334.247,Z 456.471,A -85,B 0,C 180,E1 -14870.861,E2 -14870.861} C_VEL
LIN {X 0,Y 334.967,Z 443.438,A -85,B 0,C 180,E1 -14871.338,E2 -14871.338} C_VEL
LIN {X 0,Y 336.245,Z 376.264,A -85,B 0,C 180,E1 -14872.784,E2 -14872.784} C_VEL
LIN {X 0,Y 331.234,Z 340.009,A -85,B 0,C 180,E1 -14873.98,E2 -14873.98} C_VEL
LIN {X 0,Y 329.625,Z 329.517,A -85,B 0,C 180,E1 -14874.386,E2 -14874.386} C_VEL
LIN {X 0,Y 330.261,Z 323.506,A -85,B 0,C 180,E1 -14875.863,E2 -14875.863} C_VEL
LIN {X 0,Y 328.767,Z 315.14,A -85,B 0,C 180,E1 -14878.052,E2 -14878.052} C_VEL
LIN {X 0,Y 326.651,Z 304.794,A -85,B 0,C 180,E1 -14880.872,E2 -14880.872} C_VEL
LIN {X 0,Y 326.603,Z 304.803,A -85,B 0,C 180,E1 -14884.018,E2 -14884.018} C_VEL
LIN {X 0,Y 326.623,Z 304.796,A -85,B 0,C 180,E1 -14887.237,E2 -14887.237} C_VEL
LIN {X 0,Y 326.571,Z 304.802,A -85,B 0,C 180,E1 -14891.13,E2 -14891.13} C_VEL
LIN {X 0,Y 326.522,Z 304.808,A -85,B 0,C 180,E1 -14894.742,E2 -14894.742} C_VEL
LIN {X 0,Y 326.556,Z 304.806,A -85,B 0,C 180,E1 -14898.151,E2 -14898.151} C_VEL
LIN {X 0,Y 326.561,Z 304.803,A -85,B 0,C 180,E1 -14901.382,E2 -14901.382} C_VEL
LIN {X 0,Y 326.612,Z 304.796,A -85,B 0,C 180,E1 -14904.851,E2 -14904.851} C_VEL
LIN {X 0,Y 326.6,Z 304.803,A -85,B 0,C 180,E1 -14907.455,E2 -14907.455} C_VEL
LIN {X 0,Y 326.573,Z 304.802,A -85,B 0,C 180,E1 -14910.332,E2 -14910.332} C_VEL
LIN {X 0,Y 326.589,Z 304.803,A -85,B 0,C 180,E1 -14913.134,E2 -14913.134} C_VEL
LIN {X 0,Y 326.603,Z 304.801,A -85,B 0,C 180,E1 -14915.867,E2 -14915.867} C_VEL
LIN {X 0,Y 326.613,Z 304.796,A -85,B 0,C 180,E1 -14919.862,E2 -14919.862} C_VEL
LIN {X 0,Y 326.7,Z 304.784,A -85,B 0,C 180,E1 -14923.76,E2 -14923.76} C_VEL
LIN {X 0,Y 326.75,Z 304.779,A -85,B 0,C 180,E1 -14926.314,E2 -14926.314} C_VEL
LIN {X 0,Y 326.774,Z 304.776,A -85,B 0,C 180,E1 -14930.093,E2 -14930.093} C_VEL
LIN {X 0,Y 326.929,Z 304.747,A -85,B 0,C 180,E1 -14933.83,E2 -14933.83} C_VEL
LIN {X 0,Y 327.002,Z 304.75,A -85,B 0,C 180,E1 -14937.536,E2 -14937.536} C_VEL
LIN {X 0,Y 327.036,Z 304.749,A -85,B 0,C 180,E1 -14941.231,E2 -14941.231} C_VEL
LIN {X 0,Y 326.736,Z 304.781,A -85,B 0,C 180,E1 -14943.7,E2 -14943.7} C_VEL
LIN {X 0,Y 326.905,Z 304.76,A -85,B 0,C 180,E1 -14946.574,E2 -14946.574} C_VEL
LIN {X 0,Y 326.774,Z 304.775,A -85,B 0,C 180,E1 -14949.908,E2 -14949.908} C_VEL
LIN {X 0,Y 326.751,Z 304.781,A -85,B 0,C 180,E1 -14953.686,E2 -14953.686} C_VEL
LIN {X 0,Y 326.655,Z 304.789,A -85,B 0,C 180,E1 -14957.53,E2 -14957.53} C_VEL
LIN {X 0,Y 326.623,Z 304.797,A -85,B 0,C 180,E1 -14960.138,E2 -14960.138} C_VEL
LIN {X 0,Y 326.635,Z 304.793,A -85,B 0,C 180,E1 -14964.13,E2 -14964.13} C_VEL
LIN {X 0,Y 326.62,Z 304.798,A -85,B 0,C 180,E1 -14968.254,E2 -14968.254} C_VEL
LIN {X 0,Y 326.567,Z 304.802,A -85,B 0,C 180,E1 -14971.098,E2 -14971.098} C_VEL
LIN {X 0,Y 326.6,Z 304.799,A -85,B 0,C 180,E1 -14974.02,E2 -14974.02} C_VEL
LIN {X 0,Y 326.621,Z 304.795,A -85,B 0,C 180,E1 -14977.239,E2 -14977.239} C_VEL
LIN {X 0,Y 326.571,Z 304.803,A -85,B 0,C 180,E1 -14981.132,E2 -14981.132} C_VEL
LIN {X 0,Y 326.522,Z 304.812,A -85,B 0,C 180,E1 -14984.744,E2 -14984.744} C_VEL
LIN {X 0,Y 326.572,Z 304.805,A -85,B 0,C 180,E1 -14988.156,E2 -14988.156} C_VEL
LIN {X 0,Y 326.619,Z 304.795,A -85,B 0,C 180,E1 -14991.393,E2 -14991.393} C_VEL
LIN {X 0,Y 326.616,Z 304.799,A -85,B 0,C 180,E1 -14994.853,E2 -14994.853} C_VEL
LIN {X 0,Y 326.605,Z 304.797,A -85,B 0,C 180,E1 -14997.457,E2 -14997.457} C_VEL
LIN {X 0,Y 326.645,Z 304.798,A -85,B 0,C 180,E1 -15000.341,E2 -15000.341} C_VEL
LIN {X 0,Y 326.689,Z 304.789,A -85,B 0,C 180,E1 -15004.518,E2 -15004.518} C_VEL
LIN {X 0,Y 326.698,Z 304.786,A -85,B 0,C 180,E1 -15005.268,E2 -15005.268} C_VEL
LIN {X 0,Y 327.655,Z 307.615,A -85,B 0,C 180,E1 -15005.421,E2 -15005.421} C_VEL
LIN {X 0,Y 336.018,Z 326.147,A -85,B 0,C 180,E1 -15006.505,E2 -15006.505} C_VEL
LIN {X 0,Y 337.454,Z 329.636,A -85,B 0,C 180,E1 -15006.692,E2 -15006.692} C_VEL
LIN {X 0,Y 337.641,Z 334.912,A -85,B 0,C 180,E1 -15006.826,E2 -15006.826} C_VEL
LIN {X 0,Y 335.931,Z 415.37,A -85,B 0,C 180,E1 -15008.565,E2 -15008.565} C_VEL
LIN {X 0,Y 335.442,Z 428.055,A -85,B 0,C 180,E1 -15009.056,E2 -15009.056} C_VEL
LIN {X 0,Y 334.53,Z 440.836,A -85,B 0,C 180,E1 -15009.8,E2 -15009.8} C_VEL
LIN {X 0,Y 333.466,Z 453.045,A -85,B 0,C 180,E1 -15010.775,E2 -15010.775} C_VEL
LIN {X 0,Y 332.252,Z 464.328,A -85,B 0,C 180,E1 -15011.95,E2 -15011.95} C_VEL
LIN {X 0,Y 331.1,Z 474.861,A -85,B 0,C 180,E1 -15013.35,E2 -15013.35} C_VEL
LIN {X 0,Y 329.751,Z 484.165,A -85,B 0,C 180,E1 -15014.867,E2 -15014.867} C_VEL
LIN {X 0,Y 328.696,Z 491.781,A -85,B 0,C 180,E1 -15016.398,E2 -15016.398} C_VEL
LIN {X 0,Y 327.596,Z 499.209,A -85,B 0,C 180,E1 -15018.242,E2 -15018.242} C_VEL
LIN {X 0,Y 326.683,Z 505.172,A -85,B 0,C 180,E1 -15020.091,E2 -15020.091} C_VEL
LIN {X 0,Y 326.081,Z 509.88,A -85,B 0,C 180,E1 -15021.948,E2 -15021.948} C_VEL
LIN {X 0,Y 325.628,Z 513.479,A -85,B 0,C 180,E1 -15023.806,E2 -15023.806} C_VEL
LIN {X 0,Y 325.386,Z 515.333,A -85,B 0,C 180,E1 -15025.045,E2 -15025.045} C_VEL
LIN {X 0,Y 325.203,Z 516.749,A -85,B 0,C 180,E1 -15026.284,E2 -15026.284} C_VEL
LIN {X 0,Y 325.045,Z 518.351,A -85,B 0,C 180,E1 -15028.762,E2 -15028.762} C_VEL
LIN {X 0,Y 325.044,Z 518.583,A -85,B 0,C 180,E1 -15030.001,E2 -15030.001} C_VEL
LIN {X 0,Y 325.045,Z 518.391,A -85,B 0,C 180,E1 -15031.24,E2 -15031.24} C_VEL
LIN {X 0,Y 325.2,Z 516.843,A -85,B 0,C 180,E1 -15033.719,E2 -15033.719} C_VEL
LIN {X 0,Y 325.383,Z 515.48,A -85,B 0,C 180,E1 -15034.958,E2 -15034.958} C_VEL
LIN {X 0,Y 325.815,Z 511.995,A -85,B 0,C 180,E1 -15037.138,E2 -15037.138} C_VEL
LIN {X 0,Y 326.394,Z 507.157,A -85,B 0,C 180,E1 -15039.295,E2 -15039.295} C_VEL
LIN {X 0,Y 327.253,Z 501.712,A -85,B 0,C 180,E1 -15041.146,E2 -15041.146} C_VEL
LIN {X 0,Y 328.236,Z 494.882,A -85,B 0,C 180,E1 -15042.993,E2 -15042.993} C_VEL
LIN {X 0,Y 329.492,Z 486.318,A -85,B 0,C 180,E1 -15044.832,E2 -15044.832} C_VEL
LIN {X 0,Y 330.787,Z 477.54,A -85,B 0,C 180,E1 -15046.352,E2 -15046.352} C_VEL
LIN {X 0,Y 331.881,Z 468.013,A -85,B 0,C 180,E1 -15047.708,E2 -15047.708} C_VEL
LIN {X 0,Y 333.068,Z 457.204,A -85,B 0,C 180,E1 -15048.932,E2 -15048.932} C_VEL
LIN {X 0,Y 334.247,Z 445.312,A -85,B 0,C 180,E1 -15049.98,E2 -15049.98} C_VEL
LIN {X 0,Y 335.133,Z 432.841,A -85,B 0,C 180,E1 -15050.806,E2 -15050.806} C_VEL
LIN {X 0,Y 335.88,Z 419.61,A -85,B 0,C 180,E1 -15051.4,E2 -15051.4} C_VEL
LIN {X 0,Y 336.231,Z 405.522,A -85,B 0,C 180,E1 -15051.779,E2 -15051.779} C_VEL
LIN {X 0,Y 337.711,Z 331.432,A -85,B 0,C 180,E1 -15053.359,E2 -15053.359} C_VEL
LIN {X 0,Y 337.111,Z 328.744,A -85,B 0,C 180,E1 -15053.465,E2 -15053.465} C_VEL
LIN {X 0,Y 328.604,Z 309.644,A -85,B 0,C 180,E1 -15054.567,E2 -15054.567} C_VEL
LIN {X 0,Y 326.828,Z 305.466,A -85,B 0,C 180,E1 -15054.81,E2 -15054.81} C_VEL
LIN {X 0,Y 326.687,Z 304.788,A -85,B 0,C 180,E1 -15054.886,E2 -15054.886} C_VEL
LIN {X 0,Y 326.659,Z 304.794,A -85,B 0,C 180,E1 -15058.252,E2 -15058.252} C_VEL
LIN {X 0,Y 326.659,Z 304.795,A -85,B 0,C 180,E1 -15059.571,E2 -15059.571} C_VEL
LIN {X 0,Y 326.035,Z 304.878,A -85,B 0,C 180,E1 -15060.6,E2 -15060.6} C_VEL
LIN {X 0,Y 323.158,Z 305.234,A -85,B 0,C 180,E1 -15062.273,E2 -15062.273} C_VEL
LIN {X 0,Y 320.695,Z 305.54,A -85,B 0,C 180,E1 -15063.628,E2 -15063.628} C_VEL
LIN {X 0,Y 319.645,Z 305.667,A -85,B 0,C 180,E1 -15064.679,E2 -15064.679} C_VEL
LIN {X 0,Y 319.566,Z 305.677,A -85,B 0,C 180,E1 -15065.035,E2 -15065.035} C_VEL
LIN {X 0,Y 319.579,Z 305.678,A -85,B 0,C 180,E1 -15068.009,E2 -15068.009} C_VEL
LIN {X 0,Y 319.557,Z 305.683,A -85,B 0,C 180,E1 -15071.603,E2 -15071.603} C_VEL
LIN {X 0,Y 319.52,Z 305.675,A -85,B 0,C 180,E1 -15075.263,E2 -15075.263} C_VEL
LIN {X 0,Y 319.533,Z 305.678,A -85,B 0,C 180,E1 -15078.712,E2 -15078.712} C_VEL
LIN {X 0,Y 319.559,Z 305.676,A -85,B 0,C 180,E1 -15082.35,E2 -15082.35} C_VEL
LIN {X 0,Y 319.566,Z 305.68,A -85,B 0,C 180,E1 -15085.124,E2 -15085.124} C_VEL
LIN {X 0,Y 319.571,Z 305.675,A -85,B 0,C 180,E1 -15089.06,E2 -15089.06} C_VEL
LIN {X 0,Y 319.611,Z 305.672,A -85,B 0,C 180,E1 -15092.498,E2 -15092.498} C_VEL
LIN {X 0,Y 319.616,Z 305.668,A -85,B 0,C 180,E1 -15095.305,E2 -15095.305} C_VEL
LIN {X 0,Y 319.666,Z 305.727,A -85,B 0,C 180,E1 -15096.782,E2 -15096.782} C_VEL
LIN {X 0,Y 320.099,Z 308.169,A -85,B 0,C 180,E1 -15097.552,E2 -15097.552} C_VEL
LIN {X 0,Y 325.067,Z 327.024,A -85,B 0,C 180,E1 -15098.385,E2 -15098.385} C_VEL
LIN {X 0,Y 326.366,Z 335.008,A -85,B 0,C 180,E1 -15098.696,E2 -15098.696} C_VEL
LIN {X 0,Y 323.771,Z 417.721,A -85,B 0,C 180,E1 -15101.326,E2 -15101.326} C_VEL
LIN {X 0,Y 323.237,Z 431.621,A -85,B 0,C 180,E1 -15102.033,E2 -15102.033} C_VEL
LIN {X 0,Y 322.504,Z 443.778,A -85,B 0,C 180,E1 -15102.891,E2 -15102.891} C_VEL
LIN {X 0,Y 321.8,Z 455.954,A -85,B 0,C 180,E1 -15104.001,E2 -15104.001} C_VEL
LIN {X 0,Y 321.072,Z 466.947,A -85,B 0,C 180,E1 -15105.258,E2 -15105.258} C_VEL
LIN {X 0,Y 320.235,Z 478.062,A -85,B 0,C 180,E1 -15106.839,E2 -15106.839} C_VEL
LIN {X 0,Y 319.486,Z 487.951,A -85,B 0,C 180,E1 -15108.581,E2 -15108.581} C_VEL
LIN {X 0,Y 318.901,Z 496.624,A -85,B 0,C 180,E1 -15110.486,E2 -15110.486} C_VEL
LIN {X 0,Y 318.443,Z 503.617,A -85,B 0,C 180,E1 -15112.391,E2 -15112.391} C_VEL
LIN {X 0,Y 318.155,Z 508.751,A -85,B 0,C 180,E1 -15114.138,E2 -15114.138} C_VEL
LIN {X 0,Y 318.064,Z 513.439,A -85,B 0,C 180,E1 -15116.199,E2 -15116.199} C_VEL
LIN {X 0,Y 317.93,Z 515.657,A -85,B 0,C 180,E1 -15117.466,E2 -15117.466} C_VEL
LIN {X 0,Y 317.879,Z 517.433,A -85,B 0,C 180,E1 -15118.733,E2 -15118.733} C_VEL
LIN {X 0,Y 317.906,Z 518.732,A -85,B 0,C 180,E1 -15120,E2 -15120} C_VEL
LIN {X 0,Y 318.008,Z 519.584,A -85,B 0,C 180,E1 -15121.266,E2 -15121.266} C_VEL
LIN {X 0,Y 318.176,Z 520.023,A -85,B 0,C 180,E1 -15122.532,E2 -15122.532} C_VEL
LIN {X 0,Y 318.392,Z 520.032,A -85,B 0,C 180,E1 -15123.797,E2 -15123.797} C_VEL
LIN {X 0,Y 318.526,Z 519.586,A -85,B 0,C 180,E1 -15125.063,E2 -15125.063} C_VEL
LIN {X 0,Y 318.784,Z 518.725,A -85,B 0,C 180,E1 -15126.329,E2 -15126.329} C_VEL
LIN {X 0,Y 319.599,Z 516.513,A -85,B 0,C 180,E1 -15128.283,E2 -15128.283} C_VEL
LIN {X 0,Y 320.5,Z 513.459,A -85,B 0,C 180,E1 -15130.103,E2 -15130.103} C_VEL
LIN {X 0,Y 321.613,Z 509.24,A -85,B 0,C 180,E1 -15131.982,E2 -15131.982} C_VEL
LIN {X 0,Y 322.99,Z 503.823,A -85,B 0,C 180,E1 -15133.848,E2 -15133.848} C_VEL
LIN {X 0,Y 324.652,Z 497.071,A -85,B 0,C 180,E1 -15135.7,E2 -15135.7} C_VEL
LIN {X 0,Y 326.616,Z 488.628,A -85,B 0,C 180,E1 -15137.533,E2 -15137.533} C_VEL
LIN {X 0,Y 328.542,Z 480.069,A -85,B 0,C 180,E1 -15139.04,E2 -15139.04} C_VEL
LIN {X 0,Y 330.789,Z 469.393,A -85,B 0,C 180,E1 -15140.56,E2 -15140.56} C_VEL
LIN {X 0,Y 332.72,Z 458.152,A -85,B 0,C 180,E1 -15141.856,E2 -15141.856} C_VEL
LIN {X 0,Y 334.514,Z 447.05,A -85,B 0,C 180,E1 -15142.872,E2 -15142.872} C_VEL
LIN {X 0,Y 336.185,Z 433.875,A -85,B 0,C 180,E1 -15143.812,E2 -15143.812} C_VEL
LIN {X 0,Y 337.629,Z 420.15,A -85,B 0,C 180,E1 -15144.52,E2 -15144.52} C_VEL
LIN {X 0,Y 343.874,Z 351.053,A -85,B 0,C 180,E1 -15147.084,E2 -15147.084} C_VEL
LIN {X 0,Y 339.943,Z 343.071,A -85,B 0,C 180,E1 -15148.304,E2 -15148.304} C_VEL
LIN {X 0,Y 335.682,Z 335.762,A -85,B 0,C 180,E1 -15149.701,E2 -15149.701} C_VEL
LIN {X 0,Y 333.142,Z 331.874,A -85,B 0,C 180,E1 -15150.594,E2 -15150.594} C_VEL
LIN {X 0,Y 330.472,Z 327.983,A -85,B 0,C 180,E1 -15151.607,E2 -15151.607} C_VEL
LIN {X 0,Y 327.167,Z 323.432,A -85,B 0,C 180,E1 -15152.997,E2 -15152.997} C_VEL
LIN {X 0,Y 324.133,Z 319.649,A -85,B 0,C 180,E1 -15154.44,E2 -15154.44} C_VEL
LIN {X 0,Y 323.779,Z 318.958,A -85,B 0,C 180,E1 -15154.735,E2 -15154.735} C_VEL
LIN {X 0,Y 323.265,Z 317.096,A -85,B 0,C 180,E1 -15157.499,E2 -15157.499} C_VEL
LIN {X 0,Y 322.946,Z 316.082,A -85,B 0,C 180,E1 -15160.758,E2 -15160.758} C_VEL
LIN {X 0,Y 323.111,Z 316.338,A -85,B 0,C 180,E1 -15164.127,E2 -15164.127} C_VEL
LIN {X 0,Y 323.375,Z 317.046,A -85,B 0,C 180,E1 -15165.934,E2 -15165.934} C_VEL
LIN {X 0,Y 324.114,Z 319.653,A -85,B 0,C 180,E1 -15169.418,E2 -15169.418} C_VEL
LIN {X 0,Y 325.417,Z 323.544,A -85,B 0,C 180,E1 -15172.79,E2 -15172.79} C_VEL
LIN {X 0,Y 326.7,Z 328.759,A -85,B 0,C 180,E1 -15175.99,E2 -15175.99} C_VEL
LIN {X 0,Y 327.086,Z 330.045,A -85,B 0,C 180,E1 -15176.56,E2 -15176.56} C_VEL
LIN {X 0,Y 330.197,Z 335.613,A -85,B 0,C 180,E1 -15177.916,E2 -15177.916} C_VEL
LIN {X 0,Y 331.271,Z 337.503,A -85,B 0,C 180,E1 -15178.339,E2 -15178.339} C_VEL
LIN {X 0,Y 334.34,Z 343.552,A -85,B 0,C 180,E1 -15179.524,E2 -15179.524} C_VEL
LIN {X 0,Y 336.898,Z 349.021,A -85,B 0,C 180,E1 -15180.447,E2 -15180.447} C_VEL
LIN {X 0,Y 337.784,Z 351.79,A -85,B 0,C 180,E1 -15180.801,E2 -15180.801} C_VEL
LIN {X 0,Y 340.015,Z 364.139,A -85,B 0,C 180,E1 -15181.965,E2 -15181.965} C_VEL
LIN {X 0,Y 341.577,Z 377.623,A -85,B 0,C 180,E1 -15182.984,E2 -15182.984} C_VEL
LIN {X 0,Y 341.759,Z 382.438,A -85,B 0,C 180,E1 -15183.264,E2 -15183.264} C_VEL
LIN {X 0,Y 336.206,Z 445.376,A -85,B 0,C 180,E1 -15185.574,E2 -15185.574} C_VEL
LIN {X 0,Y 334.462,Z 459.192,A -85,B 0,C 180,E1 -15186.304,E2 -15186.304} C_VEL
LIN {X 0,Y 332.524,Z 471.216,A -85,B 0,C 180,E1 -15187.146,E2 -15187.146} C_VEL
LIN {X 0,Y 330.243,Z 483.956,A -85,B 0,C 180,E1 -15188.298,E2 -15188.298} C_VEL
LIN {X 0,Y 328.01,Z 495.405,A -85,B 0,C 180,E1 -15189.623,E2 -15189.623} C_VEL
LIN {X 0,Y 325.857,Z 505.902,A -85,B 0,C 180,E1 -15191.123,E2 -15191.123} C_VEL
LIN {X 0,Y 323.652,Z 515.725,A -85,B 0,C 180,E1 -15192.86,E2 -15192.86} C_VEL
LIN {X 0,Y 321.876,Z 524.528,A -85,B 0,C 180,E1 -15194.809,E2 -15194.809} C_VEL
LIN {X 0,Y 320.427,Z 531.353,A -85,B 0,C 180,E1 -15196.684,E2 -15196.684} C_VEL
LIN {X 0,Y 319.342,Z 536.846,A -85,B 0,C 180,E1 -15198.575,E2 -15198.575} C_VEL
LIN {X 0,Y 318.567,Z 541.175,A -85,B 0,C 180,E1 -15200.475,E2 -15200.475} C_VEL
LIN {X 0,Y 318.063,Z 544.439,A -85,B 0,C 180,E1 -15202.38,E2 -15202.38} C_VEL
LIN {X 0,Y 317.838,Z 546.687,A -85,B 0,C 180,E1 -15204.29,E2 -15204.29} C_VEL
LIN {X 0,Y 317.841,Z 547.946,A -85,B 0,C 180,E1 -15206.195,E2 -15206.195} C_VEL
LIN {X 0,Y 317.815,Z 548.226,A -85,B 0,C 180,E1 -15207.464,E2 -15207.464} C_VEL
LIN {X 0,Y 317.918,Z 548.066,A -85,B 0,C 180,E1 -15208.732,E2 -15208.732} C_VEL
LIN {X 0,Y 318.121,Z 547.484,A -85,B 0,C 180,E1 -15209.999,E2 -15209.999} C_VEL
LIN {X 0,Y 317.912,Z 546.456,A -85,B 0,C 180,E1 -15212.533,E2 -15212.533} C_VEL
LIN {X 0,Y 317.911,Z 545.437,A -85,B 0,C 180,E1 -15213.801,E2 -15213.801} C_VEL
LIN {X 0,Y 317.897,Z 542.934,A -85,B 0,C 180,E1 -15215.815,E2 -15215.815} C_VEL
LIN {X 0,Y 318.032,Z 539.735,A -85,B 0,C 180,E1 -15217.618,E2 -15217.618} C_VEL
LIN {X 0,Y 318.355,Z 535.289,A -85,B 0,C 180,E1 -15219.529,E2 -15219.529} C_VEL
LIN {X 0,Y 319.071,Z 528.523,A -85,B 0,C 180,E1 -15221.755,E2 -15221.755} C_VEL
LIN {X 0,Y 320.129,Z 521.151,A -85,B 0,C 180,E1 -15223.649,E2 -15223.649} C_VEL
LIN {X 0,Y 321.399,Z 512.274,A -85,B 0,C 180,E1 -15225.48,E2 -15225.48} C_VEL
LIN {X 0,Y 322.583,Z 502.396,A -85,B 0,C 180,E1 -15227.103,E2 -15227.103} C_VEL
LIN {X 0,Y 323.994,Z 491.779,A -85,B 0,C 180,E1 -15228.495,E2 -15228.495} C_VEL
LIN {X 0,Y 325.287,Z 481.501,A -85,B 0,C 180,E1 -15229.564,E2 -15229.564} C_VEL
LIN {X 0,Y 326.555,Z 469.157,A -85,B 0,C 180,E1 -15230.551,E2 -15230.551} C_VEL
LIN {X 0,Y 327.636,Z 456.185,A -85,B 0,C 180,E1 -15231.303,E2 -15231.303} C_VEL
LIN {X 0,Y 328.367,Z 443.189,A -85,B 0,C 180,E1 -15231.789,E2 -15231.789} C_VEL
LIN {X 0,Y 329.68,Z 377.065,A -85,B 0,C 180,E1 -15233.241,E2 -15233.241} C_VEL
LIN {X 0,Y 324.822,Z 341.406,A -85,B 0,C 180,E1 -15234.446,E2 -15234.446} C_VEL
LIN {X 0,Y 322.784,Z 328.426,A -85,B 0,C 180,E1 -15234.933,E2 -15234.933} C_VEL
LIN {X 0,Y 323.194,Z 325.055,A -85,B 0,C 180,E1 -15235.778,E2 -15235.778} C_VEL
LIN {X 0,Y 322.759,Z 321.253,A -85,B 0,C 180,E1 -15236.777,E2 -15236.777} C_VEL
LIN {X 0,Y 319.889,Z 307.063,A -85,B 0,C 180,E1 -15240.643,E2 -15240.643} C_VEL
LIN {X 0,Y 319.601,Z 305.673,A -85,B 0,C 180,E1 -15241.091,E2 -15241.091} C_VEL
LIN {X 0,Y 319.556,Z 305.677,A -85,B 0,C 180,E1 -15244.875,E2 -15244.875} C_VEL
LIN {X 0,Y 319.568,Z 305.68,A -85,B 0,C 180,E1 -15248.007,E2 -15248.007} C_VEL
LIN {X 0,Y 319.519,Z 305.683,A -85,B 0,C 180,E1 -15251.595,E2 -15251.595} C_VEL
LIN {X 0,Y 319.482,Z 305.686,A -85,B 0,C 180,E1 -15255.256,E2 -15255.256} C_VEL
LIN {X 0,Y 319.498,Z 305.684,A -85,B 0,C 180,E1 -15258.406,E2 -15258.406} C_VEL
LIN {X 0,Y 319.535,Z 305.68,A -85,B 0,C 180,E1 -15262.352,E2 -15262.352} C_VEL
LIN {X 0,Y 319.553,Z 305.676,A -85,B 0,C 180,E1 -15265.122,E2 -15265.122} C_VEL
LIN {X 0,Y 319.516,Z 305.682,A -85,B 0,C 180,E1 -15268.136,E2 -15268.136} C_VEL
LIN {X 0,Y 319.556,Z 305.682,A -85,B 0,C 180,E1 -15271.605,E2 -15271.605} C_VEL
LIN {X 0,Y 319.533,Z 305.68,A -85,B 0,C 180,E1 -15275.298,E2 -15275.298} C_VEL
LIN {X 0,Y 319.557,Z 305.677,A -85,B 0,C 180,E1 -15278.045,E2 -15278.045} C_VEL
LIN {X 0,Y 319.605,Z 305.659,A -85,B 0,C 180,E1 -15282.07,E2 -15282.07} C_VEL
LIN {X 0,Y 319.724,Z 305.655,A -85,B 0,C 180,E1 -15286.007,E2 -15286.007} C_VEL
LIN {X 0,Y 319.726,Z 305.655,A -85,B 0,C 180,E1 -15289.872,E2 -15289.872} C_VEL
LIN {X 0,Y 319.887,Z 305.623,A -85,B 0,C 180,E1 -15293.693,E2 -15293.693} C_VEL
LIN {X 0,Y 319.949,Z 305.629,A -85,B 0,C 180,E1 -15297.482,E2 -15297.482} C_VEL
LIN {X 0,Y 320.003,Z 305.624,A -85,B 0,C 180,E1 -15301.259,E2 -15301.259} C_VEL
LIN {X 0,Y 319.703,Z 305.661,A -85,B 0,C 180,E1 -15305.045,E2 -15305.045} C_VEL
LIN {X 0,Y 319.843,Z 305.641,A -85,B 0,C 180,E1 -15307.576,E2 -15307.576} C_VEL
LIN {X 0,Y 319.706,Z 305.66,A -85,B 0,C 180,E1 -15311.411,E2 -15311.411} C_VEL
LIN {X 0,Y 319.704,Z 305.662,A -85,B 0,C 180,E1 -15314.711,E2 -15314.711} C_VEL
LIN {X 0,Y 319.632,Z 305.671,A -85,B 0,C 180,E1 -15319.013,E2 -15319.013} C_VEL
LIN {X 0,Y 319.55,Z 305.676,A -85,B 0,C 180,E1 -15323.321,E2 -15323.321} C_VEL
LIN {X 0,Y 319.571,Z 305.672,A -85,B 0,C 180,E1 -15326.094,E2 -15326.094} C_VEL
LIN {X 0,Y 319.551,Z 305.68,A -85,B 0,C 180,E1 -15328.938,E2 -15328.938} C_VEL
LIN {X 0,Y 319.517,Z 305.678,A -85,B 0,C 180,E1 -15331.864,E2 -15331.864} C_VEL
LIN {X 0,Y 319.573,Z 305.675,A -85,B 0,C 180,E1 -15335.544,E2 -15335.544} C_VEL
LIN {X 0,Y 319.551,Z 305.676,A -85,B 0,C 180,E1 -15338.011,E2 -15338.011} C_VEL
LIN {X 0,Y 319.52,Z 305.681,A -85,B 0,C 180,E1 -15341.598,E2 -15341.598} C_VEL
LIN {X 0,Y 319.483,Z 305.686,A -85,B 0,C 180,E1 -15345.258,E2 -15345.258} C_VEL
LIN {X 0,Y 319.524,Z 305.684,A -85,B 0,C 180,E1 -15348.713,E2 -15348.713} C_VEL
LIN {X 0,Y 319.557,Z 305.673,A -85,B 0,C 180,E1 -15352.349,E2 -15352.349} C_VEL
LIN {X 0,Y 319.557,Z 305.677,A -85,B 0,C 180,E1 -15355.125,E2 -15355.125} C_VEL
LIN {X 0,Y 319.564,Z 305.675,A -85,B 0,C 180,E1 -15359.061,E2 -15359.061} C_VEL
LIN {X 0,Y 319.604,Z 305.673,A -85,B 0,C 180,E1 -15362.499,E2 -15362.499} C_VEL
LIN {X 0,Y 319.641,Z 305.666,A -85,B 0,C 180,E1 -15364.699,E2 -15364.699} C_VEL
LIN {X 0,Y 320.774,Z 308.719,A -85,B 0,C 180,E1 -15364.879,E2 -15364.879} C_VEL
LIN {X 0,Y 329.445,Z 327.854,A -85,B 0,C 180,E1 -15366.042,E2 -15366.042} C_VEL
LIN {X 0,Y 331.186,Z 332.498,A -85,B 0,C 180,E1 -15366.285,E2 -15366.285} C_VEL
LIN {X 0,Y 329.35,Z 415.629,A -85,B 0,C 180,E1 -15368.115,E2 -15368.115} C_VEL
LIN {X 0,Y 328.845,Z 428.34,A -85,B 0,C 180,E1 -15368.615,E2 -15368.615} C_VEL
LIN {X 0,Y 327.9,Z 441.135,A -85,B 0,C 180,E1 -15369.373,E2 -15369.373} C_VEL
LIN {X 0,Y 326.784,Z 453.35,A -85,B 0,C 180,E1 -15370.366,E2 -15370.366} C_VEL
LIN {X 0,Y 325.639,Z 463.874,A -85,B 0,C 180,E1 -15371.472,E2 -15371.472} C_VEL
LIN {X 0,Y 324.456,Z 474.137,A -85,B 0,C 180,E1 -15372.836,E2 -15372.836} C_VEL
LIN {X 0,Y 322.921,Z 484.479,A -85,B 0,C 180,E1 -15374.539,E2 -15374.539} C_VEL
LIN {X 0,Y 321.783,Z 492.097,A -85,B 0,C 180,E1 -15376.1,E2 -15376.1} C_VEL
LIN {X 0,Y 320.639,Z 499.525,A -85,B 0,C 180,E1 -15377.983,E2 -15377.983} C_VEL
LIN {X 0,Y 319.707,Z 505.488,A -85,B 0,C 180,E1 -15379.873,E2 -15379.873} C_VEL
LIN {X 0,Y 319.048,Z 510.198,A -85,B 0,C 180,E1 -15381.769,E2 -15381.769} C_VEL
LIN {X 0,Y 318.582,Z 513.796,A -85,B 0,C 180,E1 -15383.669,E2 -15383.669} C_VEL
LIN {X 0,Y 318.336,Z 515.65,A -85,B 0,C 180,E1 -15384.935,E2 -15384.935} C_VEL
LIN {X 0,Y 318.132,Z 517.066,A -85,B 0,C 180,E1 -15386.201,E2 -15386.201} C_VEL
LIN {X 0,Y 317.954,Z 518.668,A -85,B 0,C 180,E1 -15388.735,E2 -15388.735} C_VEL
LIN {X 0,Y 317.951,Z 518.9,A -85,B 0,C 180,E1 -15390.001,E2 -15390.001} C_VEL
LIN {X 0,Y 317.953,Z 518.708,A -85,B 0,C 180,E1 -15391.268,E2 -15391.268} C_VEL
LIN {X 0,Y 318.129,Z 517.159,A -85,B 0,C 180,E1 -15393.801,E2 -15393.801} C_VEL
LIN {X 0,Y 318.333,Z 515.795,A -85,B 0,C 180,E1 -15395.068,E2 -15395.068} C_VEL
LIN {X 0,Y 318.756,Z 512.546,A -85,B 0,C 180,E1 -15397.172,E2 -15397.172} C_VEL
LIN {X 0,Y 319.391,Z 507.471,A -85,B 0,C 180,E1 -15399.5,E2 -15399.5} C_VEL
LIN {X 0,Y 320.306,Z 502.025,A -85,B 0,C 180,E1 -15401.39,E2 -15401.39} C_VEL
LIN {X 0,Y 321.335,Z 495.193,A -85,B 0,C 180,E1 -15403.278,E2 -15403.278} C_VEL
LIN {X 0,Y 322.647,Z 486.627,A -85,B 0,C 180,E1 -15405.154,E2 -15405.154} C_VEL
LIN {X 0,Y 323.997,Z 477.846,A -85,B 0,C 180,E1 -15406.704,E2 -15406.704} C_VEL
LIN {X 0,Y 325.257,Z 467.45,A -85,B 0,C 180,E1 -15408.195,E2 -15408.195} C_VEL
LIN {X 0,Y 326.546,Z 455.979,A -85,B 0,C 180,E1 -15409.488,E2 -15409.488} C_VEL
LIN {X 0,Y 327.599,Z 445.6,A -85,B 0,C 180,E1 -15410.404,E2 -15410.404} C_VEL
LIN {X 0,Y 328.511,Z 433.112,A -85,B 0,C 180,E1 -15411.246,E2 -15411.246} C_VEL
LIN {X 0,Y 329.297,Z 419.852,A -85,B 0,C 180,E1 -15411.85,E2 -15411.85} C_VEL
LIN {X 0,Y 329.665,Z 405.704,A -85,B 0,C 180,E1 -15412.236,E2 -15412.236} C_VEL
LIN {X 0,Y 331.245,Z 332.587,A -85,B 0,C 180,E1 -15413.82,E2 -15413.82} C_VEL
LIN {X 0,Y 326.314,Z 320.552,A -85,B 0,C 180,E1 -15414.493,E2 -15414.493} C_VEL
LIN {X 0,Y 319.78,Z 306.408,A -85,B 0,C 180,E1 -15415.377,E2 -15415.377} C_VEL
LIN {X 0,Y 319.66,Z 305.665,A -85,B 0,C 180,E1 -15415.432,E2 -15415.432} C_VEL
LIN {X 0,Y 319.593,Z 305.673,A -85,B 0,C 180,E1 -15418.934,E2 -15418.934} C_VEL
LIN {X 0,Y 319.538,Z 305.684,A -85,B 0,C 180,E1 -15421.862,E2 -15421.862} C_VEL
LIN {X 0,Y 319.566,Z 305.677,A -85,B 0,C 180,E1 -15425.035,E2 -15425.035} C_VEL
LIN {X 0,Y 318.912,Z 305.763,A -85,B 0,C 180,E1 -15426.087,E2 -15426.087} C_VEL
LIN {X 0,Y 316.053,Z 306.119,A -85,B 0,C 180,E1 -15427.799,E2 -15427.799} C_VEL
LIN {X 0,Y 313.62,Z 306.422,A -85,B 0,C 180,E1 -15429.187,E2 -15429.187} C_VEL
LIN {X 0,Y 312.578,Z 306.548,A -85,B 0,C 180,E1 -15430.262,E2 -15430.262} C_VEL
LIN {X 0,Y 312.495,Z 306.558,A -85,B 0,C 180,E1 -15430.626,E2 -15430.626} C_VEL
LIN {X 0,Y 312.477,Z 306.555,A -85,B 0,C 180,E1 -15434.206,E2 -15434.206} C_VEL
LIN {X 0,Y 312.491,Z 306.555,A -85,B 0,C 180,E1 -15437.919,E2 -15437.919} C_VEL
LIN {X 0,Y 312.504,Z 306.56,A -85,B 0,C 180,E1 -15440.972,E2 -15440.972} C_VEL
LIN {X 0,Y 312.537,Z 306.549,A -85,B 0,C 180,E1 -15444.221,E2 -15444.221} C_VEL
LIN {X 0,Y 312.509,Z 306.556,A -85,B 0,C 180,E1 -15447.334,E2 -15447.334} C_VEL
LIN {X 0,Y 312.55,Z 306.552,A -85,B 0,C 180,E1 -15451.279,E2 -15451.279} C_VEL
LIN {X 0,Y 312.592,Z 306.546,A -85,B 0,C 180,E1 -15454.711,E2 -15454.711} C_VEL
LIN {X 0,Y 312.64,Z 306.696,A -85,B 0,C 180,E1 -15456.682,E2 -15456.682} C_VEL
LIN {X 0,Y 313.022,Z 308.799,A -85,B 0,C 180,E1 -15457.284,E2 -15457.284} C_VEL
LIN {X 0,Y 318.342,Z 328.962,A -85,B 0,C 180,E1 -15458.187,E2 -15458.187} C_VEL
LIN {X 0,Y 319.404,Z 335.611,A -85,B 0,C 180,E1 -15458.452,E2 -15458.452} C_VEL
LIN {X 0,Y 316.752,Z 417.789,A -85,B 0,C 180,E1 -15461.149,E2 -15461.149} C_VEL
LIN {X 0,Y 316.198,Z 431.682,A -85,B 0,C 180,E1 -15461.87,E2 -15461.87} C_VEL
LIN {X 0,Y 315.409,Z 444.827,A -85,B 0,C 180,E1 -15462.828,E2 -15462.828} C_VEL
LIN {X 0,Y 314.677,Z 456.899,A -85,B 0,C 180,E1 -15463.968,E2 -15463.968} C_VEL
LIN {X 0,Y 314.051,Z 466.469,A -85,B 0,C 180,E1 -15465.087,E2 -15465.087} C_VEL
LIN {X 0,Y 313.186,Z 477.72,A -85,B 0,C 180,E1 -15466.702,E2 -15466.702} C_VEL
LIN {X 0,Y 312.464,Z 486.923,A -85,B 0,C 180,E1 -15468.321,E2 -15468.321} C_VEL
LIN {X 0,Y 311.948,Z 494.552,A -85,B 0,C 180,E1 -15469.944,E2 -15469.944} C_VEL
LIN {X 0,Y 311.446,Z 501.992,A -85,B 0,C 180,E1 -15471.892,E2 -15471.892} C_VEL
LIN {X 0,Y 311.175,Z 507.298,A -85,B 0,C 180,E1 -15473.602,E2 -15473.602} C_VEL
LIN {X 0,Y 311.017,Z 511.924,A -85,B 0,C 180,E1 -15475.464,E2 -15475.464} C_VEL
LIN {X 0,Y 310.851,Z 515.613,A -85,B 0,C 180,E1 -15477.408,E2 -15477.408} C_VEL
LIN {X 0,Y 310.789,Z 517.469,A -85,B 0,C 180,E1 -15478.704,E2 -15478.704} C_VEL
LIN {X 0,Y 310.811,Z 518.893,A -85,B 0,C 180,E1 -15480,E2 -15480} C_VEL
LIN {X 0,Y 310.914,Z 519.842,A -85,B 0,C 180,E1 -15481.295,E2 -15481.295} C_VEL
LIN {X 0,Y 311.09,Z 520.358,A -85,B 0,C 180,E1 -15482.59,E2 -15482.59} C_VEL
LIN {X 0,Y 311.311,Z 520.462,A -85,B 0,C 180,E1 -15483.883,E2 -15483.883} C_VEL
LIN {X 0,Y 311.471,Z 520.149,A -85,B 0,C 180,E1 -15485.178,E2 -15485.178} C_VEL
LIN {X 0,Y 311.77,Z 519.371,A -85,B 0,C 180,E1 -15486.472,E2 -15486.472} C_VEL
LIN {X 0,Y 312.626,Z 517.35,A -85,B 0,C 180,E1 -15488.444,E2 -15488.444} C_VEL
LIN {X 0,Y 313.583,Z 514.44,A -85,B 0,C 180,E1 -15490.329,E2 -15490.329} C_VEL
LIN {X 0,Y 314.79,Z 510.397,A -85,B 0,C 180,E1 -15492.245,E2 -15492.245} C_VEL
LIN {X 0,Y 316.491,Z 504.208,A -85,B 0,C 180,E1 -15494.467,E2 -15494.467} C_VEL
LIN {X 0,Y 318.318,Z 497.465,A -85,B 0,C 180,E1 -15496.35,E2 -15496.35} C_VEL
LIN {X 0,Y 320.452,Z 489.048,A -85,B 0,C 180,E1 -15498.211,E2 -15498.211} C_VEL
LIN {X 0,Y 322.562,Z 480.509,A -85,B 0,C 180,E1 -15499.738,E2 -15499.738} C_VEL
LIN {X 0,Y 324.777,Z 470.699,A -85,B 0,C 180,E1 -15501.177,E2 -15501.177} C_VEL
LIN {X 0,Y 326.969,Z 459.041,A -85,B 0,C 180,E1 -15502.56,E2 -15502.56} C_VEL
LIN {X 0,Y 328.923,Z 447.792,A -85,B 0,C 180,E1 -15503.617,E2 -15503.617} C_VEL
LIN {X 0,Y 330.703,Z 434.876,A -85,B 0,C 180,E1 -15504.566,E2 -15504.566} C_VEL
LIN {X 0,Y 332.233,Z 421.652,A -85,B 0,C 180,E1 -15505.28,E2 -15505.28} C_VEL
LIN {X 0,Y 338.849,Z 353.944,A -85,B 0,C 180,E1 -15507.871,E2 -15507.871} C_VEL
LIN {X 0,Y 334.571,Z 345.422,A -85,B 0,C 180,E1 -15509.315,E2 -15509.315} C_VEL
LIN {X 0,Y 330.323,Z 338.257,A -85,B 0,C 180,E1 -15510.859,E2 -15510.859} C_VEL
LIN {X 0,Y 327.235,Z 333.767,A -85,B 0,C 180,E1 -15512.083,E2 -15512.083} C_VEL
LIN {X 0,Y 324.28,Z 329.563,A -85,B 0,C 180,E1 -15513.412,E2 -15513.412} C_VEL
LIN {X 0,Y 320.98,Z 325.224,A -85,B 0,C 180,E1 -15515.12,E2 -15515.12} C_VEL
LIN {X 0,Y 317.431,Z 321.196,A -85,B 0,C 180,E1 -15517.382,E2 -15517.382} C_VEL
LIN {X 0,Y 317.121,Z 320.598,A -85,B 0,C 180,E1 -15517.751,E2 -15517.751} C_VEL
LIN {X 0,Y 316.909,Z 319.859,A -85,B 0,C 180,E1 -15520.025,E2 -15520.025} C_VEL
LIN {X 0,Y 316.938,Z 319.878,A -85,B 0,C 180,E1 -15523.426,E2 -15523.426} C_VEL
LIN {X 0,Y 317.17,Z 320.385,A -85,B 0,C 180,E1 -15525.159,E2 -15525.159} C_VEL
LIN {X 0,Y 317.444,Z 321.325,A -85,B 0,C 180,E1 -15526.937,E2 -15526.937} C_VEL
LIN {X 0,Y 318.368,Z 324.477,A -85,B 0,C 180,E1 -15530.591,E2 -15530.591} C_VEL
LIN {X 0,Y 319.461,Z 328.15,A -85,B 0,C 180,E1 -15533.518,E2 -15533.518} C_VEL
LIN {X 0,Y 323.144,Z 334.628,A -85,B 0,C 180,E1 -15535.665,E2 -15535.665} C_VEL
LIN {X 0,Y 324.227,Z 336.404,A -85,B 0,C 180,E1 -15536.196,E2 -15536.196} C_VEL
LIN {X 0,Y 327.871,Z 343.108,A -85,B 0,C 180,E1 -15537.849,E2 -15537.849} C_VEL
LIN {X 0,Y 330.738,Z 348.998,A -85,B 0,C 180,E1 -15539.032,E2 -15539.032} C_VEL
LIN {X 0,Y 333.175,Z 354.486,A -85,B 0,C 180,E1 -15539.978,E2 -15539.978} C_VEL
LIN {X 0,Y 335.149,Z 366.178,A -85,B 0,C 180,E1 -15541.137,E2 -15541.137} C_VEL
LIN {X 0,Y 336.51,Z 379.122,A -85,B 0,C 180,E1 -15542.163,E2 -15542.163} C_VEL
LIN {X 0,Y 336.6,Z 384.22,A -85,B 0,C 180,E1 -15542.467,E2 -15542.467} C_VEL
LIN {X 0,Y 330.811,Z 445.035,A -85,B 0,C 180,E1 -15544.771,E2 -15544.771} C_VEL
LIN {X 0,Y 328.874,Z 459.215,A -85,B 0,C 180,E1 -15545.54,E2 -15545.54} C_VEL
LIN {X 0,Y 326.817,Z 471.034,A -85,B 0,C 180,E1 -15546.388,E2 -15546.388} C_VEL
LIN {X 0,Y 324.413,Z 483.626,A -85,B 0,C 180,E1 -15547.552,E2 -15547.552} C_VEL
LIN {X 0,Y 321.759,Z 496.151,A -85,B 0,C 180,E1 -15549.042,E2 -15549.042} C_VEL
LIN {X 0,Y 319.682,Z 505.445,A -85,B 0,C 180,E1 -15550.41,E2 -15550.41} C_VEL
LIN {X 0,Y 317.11,Z 516.157,A -85,B 0,C 180,E1 -15552.363,E2 -15552.363} C_VEL
LIN {X 0,Y 315.331,Z 524.017,A -85,B 0,C 180,E1 -15554.154,E2 -15554.154} C_VEL
LIN {X 0,Y 313.775,Z 530.837,A -85,B 0,C 180,E1 -15556.066,E2 -15556.066} C_VEL
LIN {X 0,Y 312.69,Z 535.498,A -85,B 0,C 180,E1 -15557.67,E2 -15557.67} C_VEL
LIN {X 0,Y 311.78,Z 540.025,A -85,B 0,C 180,E1 -15559.61,E2 -15559.61} C_VEL
LIN {X 0,Y 311.355,Z 542.451,A -85,B 0,C 180,E1 -15560.908,E2 -15560.908} C_VEL
LIN {X 0,Y 311.009,Z 544.386,A -85,B 0,C 180,E1 -15562.206,E2 -15562.206} C_VEL
LIN {X 0,Y 310.734,Z 546.653,A -85,B 0,C 180,E1 -15564.366,E2 -15564.366} C_VEL
LIN {X 0,Y 310.749,Z 547.627,A -85,B 0,C 180,E1 -15566.108,E2 -15566.108} C_VEL
LIN {X 0,Y 310.735,Z 547.819,A -85,B 0,C 180,E1 -15567.406,E2 -15567.406} C_VEL
LIN {X 0,Y 311.062,Z 547,A -85,B 0,C 180,E1 -15569.999,E2 -15569.999} C_VEL
LIN {X 0,Y 310.931,Z 546.768,A -85,B 0,C 180,E1 -15571.294,E2 -15571.294} C_VEL
LIN {X 0,Y 310.814,Z 545.119,A -85,B 0,C 180,E1 -15573.888,E2 -15573.888} C_VEL
LIN {X 0,Y 310.799,Z 542.886,A -85,B 0,C 180,E1 -15575.754,E2 -15575.754} C_VEL
LIN {X 0,Y 310.978,Z 539.417,A -85,B 0,C 180,E1 -15577.792,E2 -15577.792} C_VEL
LIN {X 0,Y 311.314,Z 534.97,A -85,B 0,C 180,E1 -15579.747,E2 -15579.747} C_VEL
LIN {X 0,Y 312.063,Z 528.204,A -85,B 0,C 180,E1 -15582.022,E2 -15582.022} C_VEL
LIN {X 0,Y 313.194,Z 520.834,A -85,B 0,C 180,E1 -15583.958,E2 -15583.958} C_VEL
LIN {X 0,Y 314.472,Z 512.324,A -85,B 0,C 180,E1 -15585.758,E2 -15585.758} C_VEL
LIN {X 0,Y 315.62,Z 503.147,A -85,B 0,C 180,E1 -15587.326,E2 -15587.326} C_VEL
LIN {X 0,Y 317.084,Z 492.752,A -85,B 0,C 180,E1 -15588.745,E2 -15588.745} C_VEL
LIN {X 0,Y 318.603,Z 481.195,A -85,B 0,C 180,E1 -15589.992,E2 -15589.992} C_VEL
LIN {X 0,Y 319.922,Z 468.858,A -85,B 0,C 180,E1 -15590.997,E2 -15590.997} C_VEL
LIN {X 0,Y 321.048,Z 455.899,A -85,B 0,C 180,E1 -15591.762,E2 -15591.762} C_VEL
LIN {X 0,Y 321.798,Z 443.093,A -85,B 0,C 180,E1 -15592.252,E2 -15592.252} C_VEL
LIN {X 0,Y 323.161,Z 377.937,A -85,B 0,C 180,E1 -15593.712,E2 -15593.712} C_VEL
LIN {X 0,Y 318.401,Z 342.791,A -85,B 0,C 180,E1 -15594.933,E2 -15594.933} C_VEL
LIN {X 0,Y 316.039,Z 327.086,A -85,B 0,C 180,E1 -15595.551,E2 -15595.551} C_VEL
LIN {X 0,Y 316.007,Z 323.806,A -85,B 0,C 180,E1 -15596.409,E2 -15596.409} C_VEL
LIN {X 0,Y 313.752,Z 312.532,A -85,B 0,C 180,E1 -15599.523,E2 -15599.523} C_VEL
LIN {X 0,Y 312.546,Z 306.552,A -85,B 0,C 180,E1 -15601.228,E2 -15601.228} C_VEL
LIN {X 0,Y 312.502,Z 306.558,A -85,B 0,C 180,E1 -15604.209,E2 -15604.209} C_VEL
LIN {X 0,Y 312.53,Z 306.557,A -85,B 0,C 180,E1 -15608.088,E2 -15608.088} C_VEL
LIN {X 0,Y 312.478,Z 306.56,A -85,B 0,C 180,E1 -15612.08,E2 -15612.08} C_VEL
LIN {X 0,Y 312.452,Z 306.562,A -85,B 0,C 180,E1 -15616.034,E2 -15616.034} C_VEL
LIN {X 0,Y 312.448,Z 306.563,A -85,B 0,C 180,E1 -15619.884,E2 -15619.884} C_VEL
LIN {X 0,Y 312.527,Z 306.552,A -85,B 0,C 180,E1 -15624.05,E2 -15624.05} C_VEL
LIN {X 0,Y 312.494,Z 306.559,A -85,B 0,C 180,E1 -15627.333,E2 -15627.333} C_VEL
LIN {X 0,Y 312.486,Z 306.559,A -85,B 0,C 180,E1 -15631.295,E2 -15631.295} C_VEL
LIN {X 0,Y 312.513,Z 306.551,A -85,B 0,C 180,E1 -15634.705,E2 -15634.705} C_VEL
LIN {X 0,Y 312.532,Z 306.557,A -85,B 0,C 180,E1 -15637.525,E2 -15637.525} C_VEL
LIN {X 0,Y 312.558,Z 306.538,A -85,B 0,C 180,E1 -15641.651,E2 -15641.651} C_VEL
LIN {X 0,Y 312.677,Z 306.535,A -85,B 0,C 180,E1 -15645.685,E2 -15645.685} C_VEL
LIN {X 0,Y 312.676,Z 306.534,A -85,B 0,C 180,E1 -15649.641,E2 -15649.641} C_VEL
LIN {X 0,Y 312.785,Z 306.513,A -85,B 0,C 180,E1 -15652.252,E2 -15652.252} C_VEL
LIN {X 0,Y 312.679,Z 306.519,A -85,B 0,C 180,E1 -15654.842,E2 -15654.842} C_VEL
LIN {X 0,Y 312.958,Z 306.498,A -85,B 0,C 180,E1 -15658.713,E2 -15658.713} C_VEL
LIN {X 0,Y 312.97,Z 306.5,A -85,B 0,C 180,E1 -15661.287,E2 -15661.287} C_VEL
LIN {X 0,Y 312.83,Z 306.515,A -85,B 0,C 180,E1 -15666.45,E2 -15666.45} C_VEL
LIN {X 0,Y 312.742,Z 306.527,A -85,B 0,C 180,E1 -15669.051,E2 -15669.051} C_VEL
LIN {X 0,Y 312.626,Z 306.545,A -85,B 0,C 180,E1 -15672.992,E2 -15672.992} C_VEL
LIN {X 0,Y 312.613,Z 306.538,A -85,B 0,C 180,E1 -15675.651,E2 -15675.651} C_VEL
LIN {X 0,Y 312.552,Z 306.549,A -85,B 0,C 180,E1 -15679.712,E2 -15679.712} C_VEL
LIN {X 0,Y 312.518,Z 306.556,A -85,B 0,C 180,E1 -15682.781,E2 -15682.781} C_VEL
LIN {X 0,Y 312.53,Z 306.548,A -85,B 0,C 180,E1 -15685.912,E2 -15685.912} C_VEL
LIN {X 0,Y 312.496,Z 306.556,A -85,B 0,C 180,E1 -15689.655,E2 -15689.655} C_VEL
LIN {X 0,Y 312.513,Z 306.553,A -85,B 0,C 180,E1 -15693.69,E2 -15693.69} C_VEL
LIN {X 0,Y 312.519,Z 306.55,A -85,B 0,C 180,E1 -15697.386,E2 -15697.386} C_VEL
LIN {X 0,Y 312.484,Z 306.561,A -85,B 0,C 180,E1 -15700.71,E2 -15700.71} C_VEL
LIN {X 0,Y 312.446,Z 306.563,A -85,B 0,C 180,E1 -15704.211,E2 -15704.211} C_VEL
LIN {X 0,Y 312.48,Z 306.557,A -85,B 0,C 180,E1 -15707.92,E2 -15707.92} C_VEL
LIN {X 0,Y 312.531,Z 306.55,A -85,B 0,C 180,E1 -15711.912,E2 -15711.912} C_VEL
LIN {X 0,Y 312.503,Z 306.558,A -85,B 0,C 180,E1 -15715.791,E2 -15715.791} C_VEL
LIN {X 0,Y 312.518,Z 306.553,A -85,B 0,C 180,E1 -15718.855,E2 -15718.855} C_VEL
LIN {X 0,Y 312.568,Z 306.549,A -85,B 0,C 180,E1 -15721.826,E2 -15721.826} C_VEL
LIN {X 0,Y 312.6,Z 306.548,A -85,B 0,C 180,E1 -15724.098,E2 -15724.098} C_VEL
LIN {X 0,Y 313.602,Z 309.378,A -85,B 0,C 180,E1 -15724.273,E2 -15724.273} C_VEL
LIN {X 0,Y 322.12,Z 327.714,A -85,B 0,C 180,E1 -15725.452,E2 -15725.452} C_VEL
LIN {X 0,Y 324.697,Z 334.368,A -85,B 0,C 180,E1 -15725.821,E2 -15725.821} C_VEL
LIN {X 0,Y 322.797,Z 415.886,A -85,B 0,C 180,E1 -15727.647,E2 -15727.647} C_VEL
LIN {X 0,Y 322.255,Z 428.624,A -85,B 0,C 180,E1 -15728.156,E2 -15728.156} C_VEL
LIN {X 0,Y 321.279,Z 441.433,A -85,B 0,C 180,E1 -15728.928,E2 -15728.928} C_VEL
LIN {X 0,Y 320.121,Z 453.655,A -85,B 0,C 180,E1 -15729.94,E2 -15729.94} C_VEL
LIN {X 0,Y 318.937,Z 463.922,A -85,B 0,C 180,E1 -15731.035,E2 -15731.035} C_VEL
LIN {X 0,Y 317.689,Z 474.45,A -85,B 0,C 180,E1 -15732.459,E2 -15732.459} C_VEL
LIN {X 0,Y 316.103,Z 484.792,A -85,B 0,C 180,E1 -15734.197,E2 -15734.197} C_VEL
LIN {X 0,Y 314.883,Z 492.413,A -85,B 0,C 180,E1 -15735.789,E2 -15735.789} C_VEL
LIN {X 0,Y 313.701,Z 499.842,A -85,B 0,C 180,E1 -15737.713,E2 -15737.713} C_VEL
LIN {X 0,Y 312.716,Z 505.806,A -85,B 0,C 180,E1 -15739.644,E2 -15739.644} C_VEL
LIN {X 0,Y 312.024,Z 510.515,A -85,B 0,C 180,E1 -15741.583,E2 -15741.583} C_VEL
LIN {X 0,Y 311.539,Z 514.113,A -85,B 0,C 180,E1 -15743.525,E2 -15743.525} C_VEL
LIN {X 0,Y 311.289,Z 515.966,A -85,B 0,C 180,E1 -15744.82,E2 -15744.82} C_VEL
LIN {X 0,Y 311.065,Z 517.382,A -85,B 0,C 180,E1 -15746.115,E2 -15746.115} C_VEL
LIN {X 0,Y 310.862,Z 518.985,A -85,B 0,C 180,E1 -15748.706,E2 -15748.706} C_VEL
LIN {X 0,Y 310.859,Z 519.217,A -85,B 0,C 180,E1 -15750.001,E2 -15750.001} C_VEL
LIN {X 0,Y 310.862,Z 519.024,A -85,B 0,C 180,E1 -15751.297,E2 -15751.297} C_VEL
LIN {X 0,Y 311.062,Z 517.475,A -85,B 0,C 180,E1 -15753.888,E2 -15753.888} C_VEL
LIN {X 0,Y 311.285,Z 516.11,A -85,B 0,C 180,E1 -15755.183,E2 -15755.183} C_VEL
LIN {X 0,Y 311.677,Z 513.15,A -85,B 0,C 180,E1 -15757.18,E2 -15757.18} C_VEL
LIN {X 0,Y 312.172,Z 509.352,A -85,B 0,C 180,E1 -15759.068,E2 -15759.068} C_VEL
LIN {X 0,Y 312.995,Z 504.302,A -85,B 0,C 180,E1 -15761.004,E2 -15761.004} C_VEL
LIN {X 0,Y 314.023,Z 497.936,A -85,B 0,C 180,E1 -15762.934,E2 -15762.934} C_VEL
LIN {X 0,Y 315.28,Z 490.009,A -85,B 0,C 180,E1 -15764.855,E2 -15764.855} C_VEL
LIN {X 0,Y 316.664,Z 481.891,A -85,B 0,C 180,E1 -15766.439,E2 -15766.439} C_VEL
LIN {X 0,Y 317.994,Z 471.92,A -85,B 0,C 180,E1 -15768.025,E2 -15768.025} C_VEL
LIN {X 0,Y 319.377,Z 460.705,A -85,B 0,C 180,E1 -15769.442,E2 -15769.442} C_VEL
LIN {X 0,Y 320.589,Z 449.67,A -85,B 0,C 180,E1 -15770.535,E2 -15770.535} C_VEL
LIN {X 0,Y 321.695,Z 437.181,A -85,B 0,C 180,E1 -15771.466,E2 -15771.466} C_VEL
LIN {X 0,Y 322.534,Z 424.1,A -85,B 0,C 180,E1 -15772.164,E2 -15772.164} C_VEL
LIN {X 0,Y 322.988,Z 411.125,A -85,B 0,C 180,E1 -15772.595,E2 -15772.595} C_VEL
LIN {X 0,Y 324.699,Z 334.716,A -85,B 0,C 180,E1 -15774.284,E2 -15774.284} C_VEL
LIN {X 0,Y 324.097,Z 332.407,A -85,B 0,C 180,E1 -15774.388,E2 -15774.388} C_VEL
LIN {X 0,Y 315.332,Z 312.796,A -85,B 0,C 180,E1 -15775.605,E2 -15775.605} C_VEL
LIN {X 0,Y 312.717,Z 307.189,A -85,B 0,C 180,E1 -15775.978,E2 -15775.978} C_VEL
LIN {X 0,Y 312.604,Z 306.544,A -85,B 0,C 180,E1 -15776.029,E2 -15776.029} C_VEL
LIN {X 0,Y 312.55,Z 306.552,A -85,B 0,C 180,E1 -15779.651,E2 -15779.651} C_VEL
LIN {X 0,Y 312.524,Z 306.558,A -85,B 0,C 180,E1 -15783.69,E2 -15783.69} C_VEL
LIN {X 0,Y 312.543,Z 306.554,A -85,B 0,C 180,E1 -15787.384,E2 -15787.384} C_VEL
LIN {X 0,Y 312.495,Z 306.558,A -85,B 0,C 180,E1 -15790.626,E2 -15790.626} C_VEL
LIN {X 0,Y 311.819,Z 306.646,A -85,B 0,C 180,E1 -15791.702,E2 -15791.702} C_VEL
LIN {X 0,Y 308.929,Z 307.001,A -85,B 0,C 180,E1 -15793.453,E2 -15793.453} C_VEL
LIN {X 0,Y 306.506,Z 307.296,A -85,B 0,C 180,E1 -15794.873,E2 -15794.873} C_VEL
LIN {X 0,Y 305.507,Z 307.414,A -85,B 0,C 180,E1 -15795.973,E2 -15795.973} C_VEL
LIN {X 0,Y 305.448,Z 307.421,A -85,B 0,C 180,E1 -15796.346,E2 -15796.346} C_VEL
LIN {X 0,Y 305.463,Z 307.434,A -85,B 0,C 180,E1 -15799.893,E2 -15799.893} C_VEL
LIN {X 0,Y 305.485,Z 307.428,A -85,B 0,C 180,E1 -15803.632,E2 -15803.632} C_VEL
LIN {X 0,Y 305.47,Z 307.433,A -85,B 0,C 180,E1 -15806.484,E2 -15806.484} C_VEL
LIN {X 0,Y 305.463,Z 307.429,A -85,B 0,C 180,E1 -15809.591,E2 -15809.591} C_VEL
LIN {X 0,Y 305.52,Z 307.429,A -85,B 0,C 180,E1 -15812.608,E2 -15812.608} C_VEL
LIN {X 0,Y 305.569,Z 307.419,A -85,B 0,C 180,E1 -15816.464,E2 -15816.464} C_VEL
LIN {X 0,Y 305.866,Z 309.053,A -85,B 0,C 180,E1 -15816.985,E2 -15816.985} C_VEL
LIN {X 0,Y 311.547,Z 330.58,A -85,B 0,C 180,E1 -15817.975,E2 -15817.975} C_VEL
LIN {X 0,Y 312.443,Z 336.452,A -85,B 0,C 180,E1 -15818.214,E2 -15818.214} C_VEL
LIN {X 0,Y 309.698,Z 418.402,A -85,B 0,C 180,E1 -15821.004,E2 -15821.004} C_VEL
LIN {X 0,Y 309.163,Z 431.494,A -85,B 0,C 180,E1 -15821.7,E2 -15821.7} C_VEL
LIN {X 0,Y 308.414,Z 443.818,A -85,B 0,C 180,E1 -15822.597,E2 -15822.597} C_VEL
LIN {X 0,Y 307.65,Z 456.338,A -85,B 0,C 180,E1 -15823.786,E2 -15823.786} C_VEL
LIN {X 0,Y 307.035,Z 465.867,A -85,B 0,C 180,E1 -15824.908,E2 -15824.908} C_VEL
LIN {X 0,Y 306.173,Z 476.294,A -85,B 0,C 180,E1 -15826.392,E2 -15826.392} C_VEL
LIN {X 0,Y 305.448,Z 485.77,A -85,B 0,C 180,E1 -15828.049,E2 -15828.049} C_VEL
LIN {X 0,Y 304.828,Z 495.078,A -85,B 0,C 180,E1 -15830.042,E2 -15830.042} C_VEL
LIN {X 0,Y 304.319,Z 502.489,A -85,B 0,C 180,E1 -15832.035,E2 -15832.035} C_VEL
LIN {X 0,Y 304.053,Z 507.516,A -85,B 0,C 180,E1 -15833.686,E2 -15833.686} C_VEL
LIN {X 0,Y 303.904,Z 513.069,A -85,B 0,C 180,E1 -15836.022,E2 -15836.022} C_VEL
LIN {X 0,Y 303.774,Z 515.539,A -85,B 0,C 180,E1 -15837.348,E2 -15837.348} C_VEL
LIN {X 0,Y 303.702,Z 517.483,A -85,B 0,C 180,E1 -15838.674,E2 -15838.674} C_VEL
LIN {X 0,Y 303.719,Z 518.991,A -85,B 0,C 180,E1 -15840,E2 -15840} C_VEL
LIN {X 0,Y 303.824,Z 520.075,A -85,B 0,C 180,E1 -15841.325,E2 -15841.325} C_VEL
LIN {X 0,Y 304.006,Z 520.691,A -85,B 0,C 180,E1 -15842.65,E2 -15842.65} C_VEL
LIN {X 0,Y 304.234,Z 520.878,A -85,B 0,C 180,E1 -15843.974,E2 -15843.974} C_VEL
LIN {X 0,Y 304.422,Z 520.663,A -85,B 0,C 180,E1 -15845.299,E2 -15845.299} C_VEL
LIN {X 0,Y 304.759,Z 520.028,A -85,B 0,C 180,E1 -15846.621,E2 -15846.621} C_VEL
LIN {X 0,Y 305.654,Z 518.203,A -85,B 0,C 180,E1 -15848.611,E2 -15848.611} C_VEL
LIN {X 0,Y 307.043,Z 514.255,A -85,B 0,C 180,E1 -15851.219,E2 -15851.219} C_VEL
LIN {X 0,Y 308.469,Z 510.037,A -85,B 0,C 180,E1 -15853.17,E2 -15853.17} C_VEL
LIN {X 0,Y 310.089,Z 504.656,A -85,B 0,C 180,E1 -15855.108,E2 -15855.108} C_VEL
LIN {X 0,Y 312.059,Z 497.948,A -85,B 0,C 180,E1 -15857.024,E2 -15857.024} C_VEL
LIN {X 0,Y 314.375,Z 489.58,A -85,B 0,C 180,E1 -15858.914,E2 -15858.914} C_VEL
LIN {X 0,Y 317.097,Z 479.232,A -85,B 0,C 180,E1 -15860.77,E2 -15860.77} C_VEL
LIN {X 0,Y 319.406,Z 469.485,A -85,B 0,C 180,E1 -15862.169,E2 -15862.169} C_VEL
LIN {X 0,Y 321.697,Z 458.188,A -85,B 0,C 180,E1 -15863.497,E2 -15863.497} C_VEL
LIN {X 0,Y 323.981,Z 445.252,A -85,B 0,C 180,E1 -15864.682,E2 -15864.682} C_VEL
LIN {X 0,Y 325.956,Z 431.628,A -85,B 0,C 180,E1 -15865.631,E2 -15865.631} C_VEL
LIN {X 0,Y 327.59,Z 416.997,A -85,B 0,C 180,E1 -15866.348,E2 -15866.348} C_VEL
LIN {X 0,Y 333.953,Z 357.022,A -85,B 0,C 180,E1 -15868.693,E2 -15868.693} C_VEL
LIN {X 0,Y 330.014,Z 349.227,A -85,B 0,C 180,E1 -15870.134,E2 -15870.134} C_VEL
LIN {X 0,Y 326.75,Z 343.595,A -85,B 0,C 180,E1 -15871.425,E2 -15871.425} C_VEL
LIN {X 0,Y 323.899,Z 339.263,A -85,B 0,C 180,E1 -15872.648,E2 -15872.648} C_VEL
LIN {X 0,Y 321.563,Z 335.835,A -85,B 0,C 180,E1 -15873.767,E2 -15873.767} C_VEL
LIN {X 0,Y 318.379,Z 331.551,A -85,B 0,C 180,E1 -15875.519,E2 -15875.519} C_VEL
LIN {X 0,Y 315.151,Z 327.581,A -85,B 0,C 180,E1 -15877.757,E2 -15877.757} C_VEL
LIN {X 0,Y 312.078,Z 325.019,A -85,B 0,C 180,E1 -15880.774,E2 -15880.774} C_VEL
LIN {X 0,Y 311.001,Z 323.726,A -85,B 0,C 180,E1 -15883.209,E2 -15883.209} C_VEL
LIN {X 0,Y 311.003,Z 323.829,A -85,B 0,C 180,E1 -15884.47,E2 -15884.47} C_VEL
LIN {X 0,Y 311.492,Z 325.544,A -85,B 0,C 180,E1 -15887.628,E2 -15887.628} C_VEL
LIN {X 0,Y 313.441,Z 329.472,A -85,B 0,C 180,E1 -15890.414,E2 -15890.414} C_VEL
LIN {X 0,Y 317.045,Z 334.742,A -85,B 0,C 180,E1 -15893.235,E2 -15893.235} C_VEL
LIN {X 0,Y 320.615,Z 341.07,A -85,B 0,C 180,E1 -15895.389,E2 -15895.389} C_VEL
LIN {X 0,Y 324.428,Z 348.47,A -85,B 0,C 180,E1 -15897.295,E2 -15897.295} C_VEL
LIN {X 0,Y 327.384,Z 354.849,A -85,B 0,C 180,E1 -15898.605,E2 -15898.605} C_VEL
LIN {X 0,Y 329.052,Z 358.857,A -85,B 0,C 180,E1 -15899.31,E2 -15899.31} C_VEL
LIN {X 0,Y 330.795,Z 371.005,A -85,B 0,C 180,E1 -15900.526,E2 -15900.526} C_VEL
LIN {X 0,Y 331.748,Z 382.585,A -85,B 0,C 180,E1 -15901.449,E2 -15901.449} C_VEL
LIN {X 0,Y 331.635,Z 385.857,A -85,B 0,C 180,E1 -15901.626,E2 -15901.626} C_VEL
LIN {X 0,Y 325.591,Z 444.492,A -85,B 0,C 180,E1 -15903.908,E2 -15903.908} C_VEL
LIN {X 0,Y 323.57,Z 458.484,A -85,B 0,C 180,E1 -15904.682,E2 -15904.682} C_VEL
LIN {X 0,Y 321.192,Z 471.158,A -85,B 0,C 180,E1 -15905.605,E2 -15905.605} C_VEL
LIN {X 0,Y 318.672,Z 483.5,A -85,B 0,C 180,E1 -15906.782,E2 -15906.782} C_VEL
LIN {X 0,Y 315.816,Z 495.908,A -85,B 0,C 180,E1 -15908.285,E2 -15908.285} C_VEL
LIN {X 0,Y 313.138,Z 506.929,A -85,B 0,C 180,E1 -15909.984,E2 -15909.984} C_VEL
LIN {X 0,Y 310.515,Z 517.021,A -85,B 0,C 180,E1 -15911.916,E2 -15911.916} C_VEL
LIN {X 0,Y 308.56,Z 524.807,A -85,B 0,C 180,E1 -15913.797,E2 -15913.797} C_VEL
LIN {X 0,Y 306.681,Z 532.33,A -85,B 0,C 180,E1 -15916.076,E2 -15916.076} C_VEL
LIN {X 0,Y 305.424,Z 537.44,A -85,B 0,C 180,E1 -15918.047,E2 -15918.047} C_VEL
LIN {X 0,Y 304.521,Z 541.419,A -85,B 0,C 180,E1 -15920.031,E2 -15920.031} C_VEL
LIN {X 0,Y 303.952,Z 544.354,A -85,B 0,C 180,E1 -15922.024,E2 -15922.024} C_VEL
LIN {X 0,Y 303.661,Z 546.581,A -85,B 0,C 180,E1 -15924.387,E2 -15924.387} C_VEL
LIN {X 0,Y 303.658,Z 547.289,A -85,B 0,C 180,E1 -15926.017,E2 -15926.017} C_VEL
